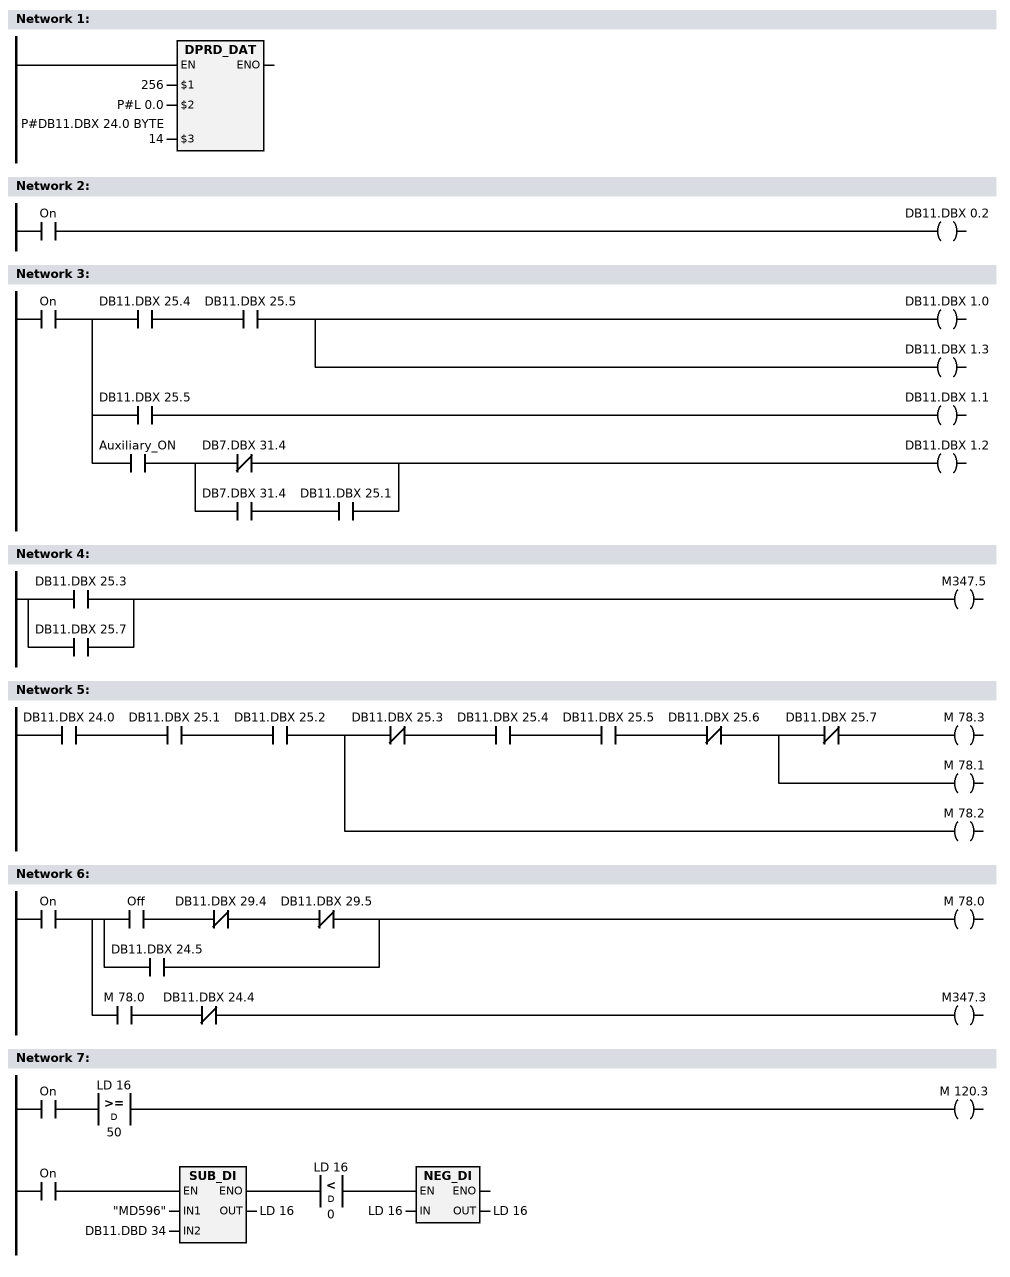
[picture p149: FC - AUTOMATIC networks 1-7]
NETWORK
TITLE =
      CALL  "DPRD_DAT" (
           $1                       := 256,
           $2                       := P#L 0.0,
           $3                       := P#DB11.DBX 24.0 BYTE 14);
      NOP   0;
NETWORK
TITLE =
      A     "On";
      =     DB11.DBX 0.2;
NETWORK
TITLE =
      A     "On";
      =     L 21.0;
      A     L 21.0;
      A     DB11.DBX 25.4;
      A     DB11.DBX 25.5;
      =     DB11.DBX 1.0;
      =     DB11.DBX 1.3;
      A     L 21.0;
      A     DB11.DBX 25.5;
      =     DB11.DBX 1.1;
      A     L 21.0;
      A     "Auxiliary_ON";
      A(;
      ON    DB7.DBX 31.4;
      O;
      A     DB7.DBX 31.4;
      A     DB11.DBX 25.1;
      );
      =     DB11.DBX 1.2;
NETWORK
TITLE =
      O     DB11.DBX 25.3;
      O     DB11.DBX 25.7;
      =     "M347.5";
NETWORK
TITLE =
      A     DB11.DBX 24.0;
      A     DB11.DBX 25.1;
      A     DB11.DBX 25.2;
      =     L 21.0;
      A     L 21.0;
      AN    DB11.DBX 25.3;
      A     DB11.DBX 25.4;
      A     DB11.DBX 25.5;
      AN    DB11.DBX 25.6;
      =     L 21.1;
      A     L 21.1;
      AN    DB11.DBX 25.7;
      =     M 78.3;
      A     L 21.1;
      BLD   102;
      =     M 78.1;
      A     L 21.0;
      BLD   102;
      =     M 78.2;
NETWORK
TITLE =
      A     "On";
      =     L 21.0;
      A     L 21.0;
      A(;
      A     "Off";
      AN    DB11.DBX 29.4;
      AN    DB11.DBX 29.5;
      O     DB11.DBX 24.5;
      );
      =     M 78.0;
      A     L 21.0;
      A     M 78.0;
      AN    DB11.DBX 24.4;
      =     "M347.3";
NETWORK
TITLE =
      A     "On";
      =     L 20.0;
      A(;
      A     L 20.0;
      JNB   M001;
      L     "MD596";
      L     DB11.DBD 34;
      -D;
      T     LD 16;
      AN    OV;
      SAVE;
      CLR;
M001: A     BR;
      );
      A(;
      L     LD 16;
      L     0;
      <D;
      );
      JNB   M002;
      L     LD 16;
      NEGD;
      T     LD 16;
M002: NOP   0;
      A     L 20.0;
      A(;
      L     LD 16;
      L     50;
      >=D;
      );
      =     M 120.3;
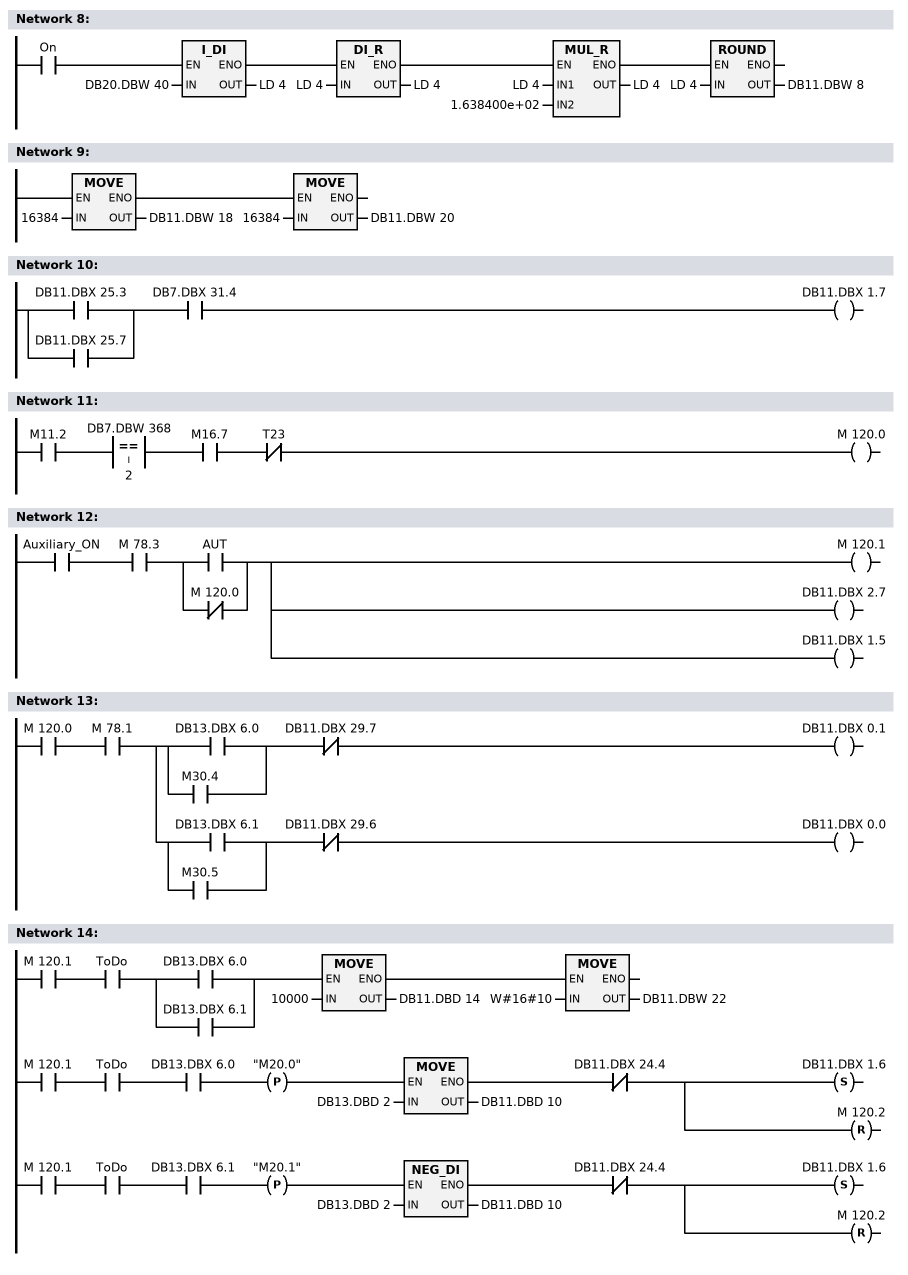
NETWORK
TITLE =
      A(;
      A(;
      A(;
      A     "On";
      JNB   M003;
      L     DB20.DBW 40;
      ITD;
      T     LD 4;
      SET;
      SAVE;
      CLR;
M003: A     BR;
      );
      JNB   M004;
      L     LD 4;
      DTR;
      T     LD 4;
      SET;
      SAVE;
      CLR;
M004: A     BR;
      );
      JNB   M005;
      L     LD 4;
      L     1.638400e+02;
      *R;
      T     LD 4;
      AN    OV;
      SAVE;
      CLR;
M005: A     BR;
      );
      JNB   M006;
      L     LD 4;
      RND;
      T     DB11.DBW 8;
M006: NOP   0;
NETWORK
TITLE =
      A(;
      L     16384;
      T     DB11.DBW 18;
      SET;
      SAVE;
      CLR;
      A     BR;
      );
      JNB   M007;
      L     16384;
      T     DB11.DBW 20;
M007: NOP   0;
NETWORK
TITLE =
      A(;
      O     DB11.DBX 25.3;
      O     DB11.DBX 25.7;
      );
      A     DB7.DBX 31.4;
      =     DB11.DBX 1.7;
NETWORK
TITLE =
      A     "M11.2";
      A(;
      L     DB7.DBW 368;
      L     2;
      ==I;
      );
      A     "M16.7";
      AN    "T23";
      =     M 120.0;
NETWORK
TITLE =
      A     "Auxiliary_ON";
      A     M 78.3;
      A(;
      O     "AUT";
      ON    M 120.0;
      );
      =     M 120.1;
      =     DB11.DBX 2.7;
      =     DB11.DBX 1.5;
NETWORK
TITLE =
      A     M 120.0;
      A     M 78.1;
      =     L 21.0;
      A     L 21.0;
      A(;
      O     DB13.DBX 6.0;
      O     "M30.4";
      );
      AN    DB11.DBX 29.7;
      =     DB11.DBX 0.1;
      A     L 21.0;
      A(;
      O     DB13.DBX 6.1;
      O     "M30.5";
      );
      AN    DB11.DBX 29.6;
      =     DB11.DBX 0.0;
NETWORK
TITLE =
      A     M 120.1;
      A     "ToDo";
      =     L 21.0;
      A(;
      A     L 21.0;
      A(;
      O     DB13.DBX 6.0;
      O     DB13.DBX 6.1;
      );
      JNB   M008;
      L     10000;
      T     DB11.DBD 14;
      SET;
      SAVE;
      CLR;
M008: A     BR;
      );
      JNB   M009;
      L     W#16#10;
      T     DB11.DBW 22;
M009: NOP   0;
      A(;
      A     L 21.0;
      A     DB13.DBX 6.0;
      FP    "M20.0";
      JNB   M010;
      L     DB13.DBD 2;
      T     DB11.DBD 10;
      SET;
      SAVE;
      CLR;
M010: A     BR;
      );
      AN    DB11.DBX 24.4;
      S     DB11.DBX 1.6;
      R     M 120.2;
      A(;
      A     L 21.0;
      A     DB13.DBX 6.1;
      FP    "M20.1";
      JNB   M011;
      L     DB13.DBD 2;
      NEGD;
      T     DB11.DBD 10;
      AN    OV;
      SAVE;
      CLR;
M011: A     BR;
      );
      AN    DB11.DBX 24.4;
      S     DB11.DBX 1.6;
      R     M 120.2;
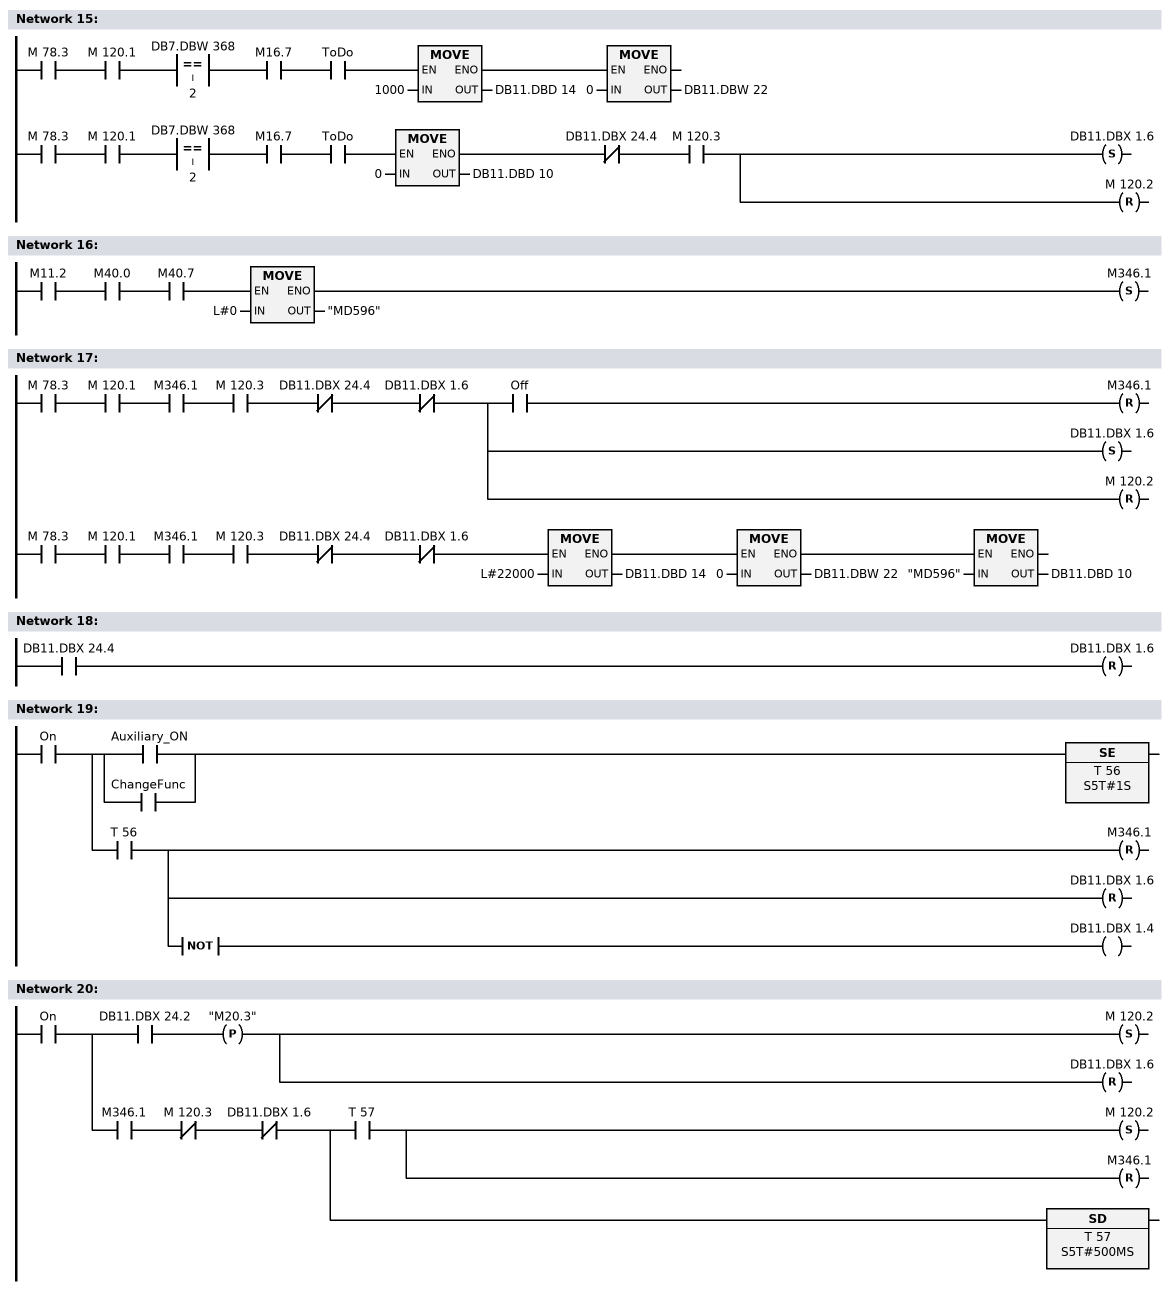
NETWORK
TITLE =
      A     M 78.3;
      A     M 120.1;
      A(;
      L     DB7.DBW 368;
      L     2;
      ==I;
      );
      A     "M16.7";
      =     L 21.0;
      A(;
      A     L 21.0;
      A     "ToDo";
      JNB   M012;
      L     1000;
      T     DB11.DBD 14;
      SET;
      SAVE;
      CLR;
M012: A     BR;
      );
      JNB   M013;
      L     0;
      T     DB11.DBW 22;
M013: NOP   0;
      A(;
      A     L 21.0;
      A     "ToDo";
      JNB   M014;
      L     0;
      T     DB11.DBD 10;
      SET;
      SAVE;
      CLR;
M014: A     BR;
      );
      AN    DB11.DBX 24.4;
      A     M 120.3;
      S     DB11.DBX 1.6;
      R     M 120.2;
NETWORK
TITLE =
      A     "M11.2";
      A     "M40.0";
      A     "M40.7";
      JNB   M015;
      L     L#0;
      T     "MD596";
      SET;
      SAVE;
      CLR;
M015: A     BR;
      S     "M346.1";
NETWORK
TITLE =
      A     M 78.3;
      A     M 120.1;
      A     "M346.1";
      A     M 120.3;
      AN    DB11.DBX 24.4;
      AN    DB11.DBX 1.6;
      =     L 21.0;
      A(;
      A(;
      A     L 21.0;
      JNB   M016;
      L     L#22000;
      T     DB11.DBD 14;
      SET;
      SAVE;
      CLR;
M016: A     BR;
      );
      JNB   M017;
      L     0;
      T     DB11.DBW 22;
      SET;
      SAVE;
      CLR;
M017: A     BR;
      );
      JNB   M018;
      L     "MD596";
      T     DB11.DBD 10;
M018: NOP   0;
      A     L 21.0;
      A     "Off";
      R     "M346.1";
      A     L 21.0;
      BLD   102;
      S     DB11.DBX 1.6;
      A     L 21.0;
      BLD   102;
      R     M 120.2;
NETWORK
TITLE =
      A     DB11.DBX 24.4;
      R     DB11.DBX 1.6;
NETWORK
TITLE =
      A     "On";
      =     L 21.0;
      A     L 21.0;
      A(;
      O     "Auxiliary_ON";
      O     "ChangeFunc";
      );
      L     S5T#1S;
      SE    T 56;
      A     L 21.0;
      A     T 56;
      =     L 21.1;
      A     L 21.1;
      BLD   102;
      R     "M346.1";
      A     L 21.1;
      BLD   102;
      R     DB11.DBX 1.6;
      A     L 21.1;
      NOT;
      =     DB11.DBX 1.4;
NETWORK
TITLE =
      A     "On";
      =     L 21.0;
      A     L 21.0;
      A     DB11.DBX 24.2;
      FP    "M20.3";
      S     M 120.2;
      R     DB11.DBX 1.6;
      A     L 21.0;
      A     "M346.1";
      AN    M 120.3;
      AN    DB11.DBX 1.6;
      =     L 21.1;
      A     L 21.1;
      A     T 57;
      S     M 120.2;
      R     "M346.1";
      A     L 21.1;
      BLD   102;
      L     S5T#500MS;
      SD    T 57;
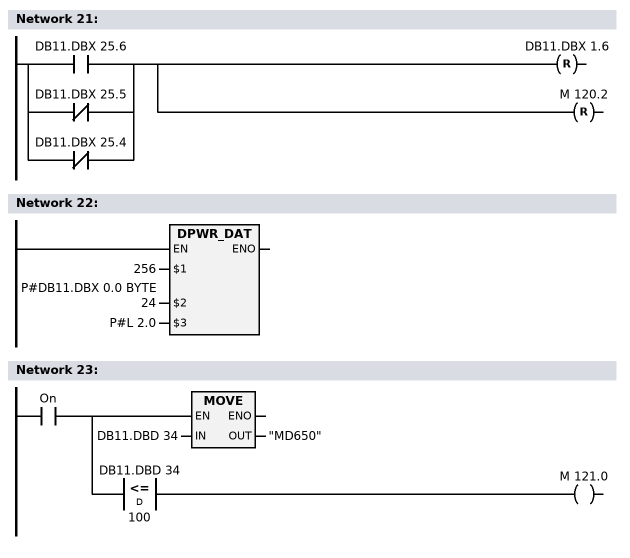
NETWORK
TITLE =
      O     DB11.DBX 25.6;
      ON    DB11.DBX 25.5;
      ON    DB11.DBX 25.4;
      R     DB11.DBX 1.6;
      R     M 120.2;
NETWORK
TITLE =
      CALL  "DPWR_DAT" (
           $1                       := 256,
           $2                       := P#DB11.DBX 0.0 BYTE 24,
           $3                       := P#L 2.0);
      NOP   0;
NETWORK
TITLE =
      A     "On";
      =     L 20.0;
      A     L 20.0;
      JNB   M019;
      L     DB11.DBD 34;
      T     "MD650";
M019: NOP   0;
      A     L 20.0;
      A(;
      L     DB11.DBD 34;
      L     100;
      <=D;
      );
      =     M 121.0;
END_FUNCTION

FUNCTION FC 25 : VOID
VERSION : 0.1
BEGIN
// (block stored without names or comments; labels and parameter names are numbered)
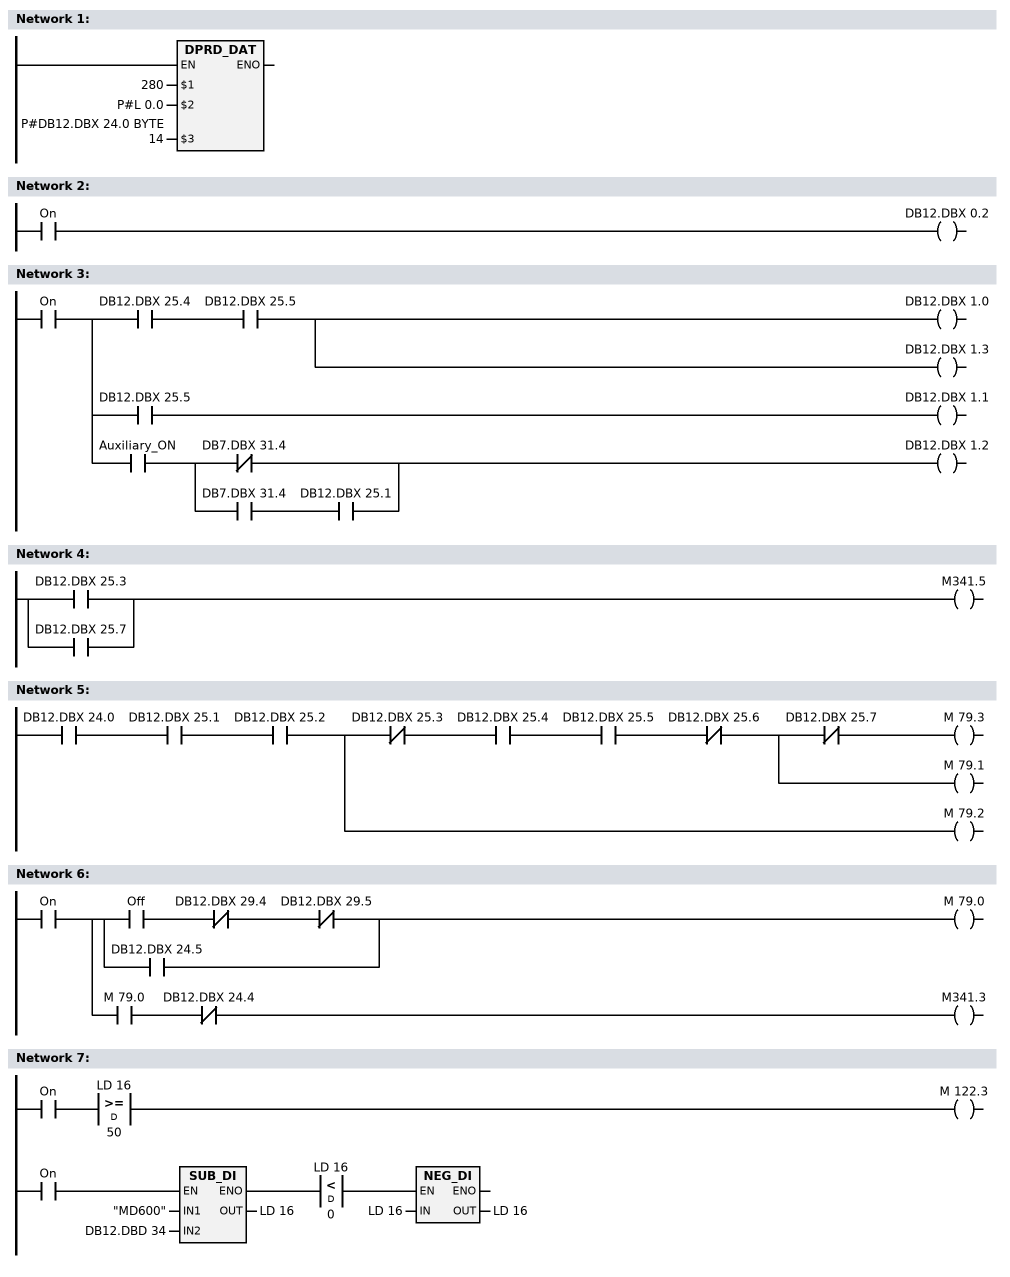
NETWORK
TITLE =
      CALL  "DPRD_DAT" (
           $1                       := 280,
           $2                       := P#L 0.0,
           $3                       := P#DB12.DBX 24.0 BYTE 14);
      NOP   0;
NETWORK
TITLE =
      A     "On";
      =     DB12.DBX 0.2;
NETWORK
TITLE =
      A     "On";
      =     L 21.0;
      A     L 21.0;
      A     DB12.DBX 25.4;
      A     DB12.DBX 25.5;
      =     DB12.DBX 1.0;
      =     DB12.DBX 1.3;
      A     L 21.0;
      A     DB12.DBX 25.5;
      =     DB12.DBX 1.1;
      A     L 21.0;
      A     "Auxiliary_ON";
      A(;
      ON    DB7.DBX 31.4;
      O;
      A     DB7.DBX 31.4;
      A     DB12.DBX 25.1;
      );
      =     DB12.DBX 1.2;
NETWORK
TITLE =
      O     DB12.DBX 25.3;
      O     DB12.DBX 25.7;
      =     "M341.5";
NETWORK
TITLE =
      A     DB12.DBX 24.0;
      A     DB12.DBX 25.1;
      A     DB12.DBX 25.2;
      =     L 21.0;
      A     L 21.0;
      AN    DB12.DBX 25.3;
      A     DB12.DBX 25.4;
      A     DB12.DBX 25.5;
      AN    DB12.DBX 25.6;
      =     L 21.1;
      A     L 21.1;
      AN    DB12.DBX 25.7;
      =     M 79.3;
      A     L 21.1;
      BLD   102;
      =     M 79.1;
      A     L 21.0;
      BLD   102;
      =     M 79.2;
NETWORK
TITLE =
      A     "On";
      =     L 21.0;
      A     L 21.0;
      A(;
      A     "Off";
      AN    DB12.DBX 29.4;
      AN    DB12.DBX 29.5;
      O     DB12.DBX 24.5;
      );
      =     M 79.0;
      A     L 21.0;
      A     M 79.0;
      AN    DB12.DBX 24.4;
      =     "M341.3";
NETWORK
TITLE =
      A     "On";
      =     L 20.0;
      A(;
      A     L 20.0;
      JNB   M001;
      L     "MD600";
      L     DB12.DBD 34;
      -D;
      T     LD 16;
      AN    OV;
      SAVE;
      CLR;
M001: A     BR;
      );
      A(;
      L     LD 16;
      L     0;
      <D;
      );
      JNB   M002;
      L     LD 16;
      NEGD;
      T     LD 16;
M002: NOP   0;
      A     L 20.0;
      A(;
      L     LD 16;
      L     50;
      >=D;
      );
      =     M 122.3;
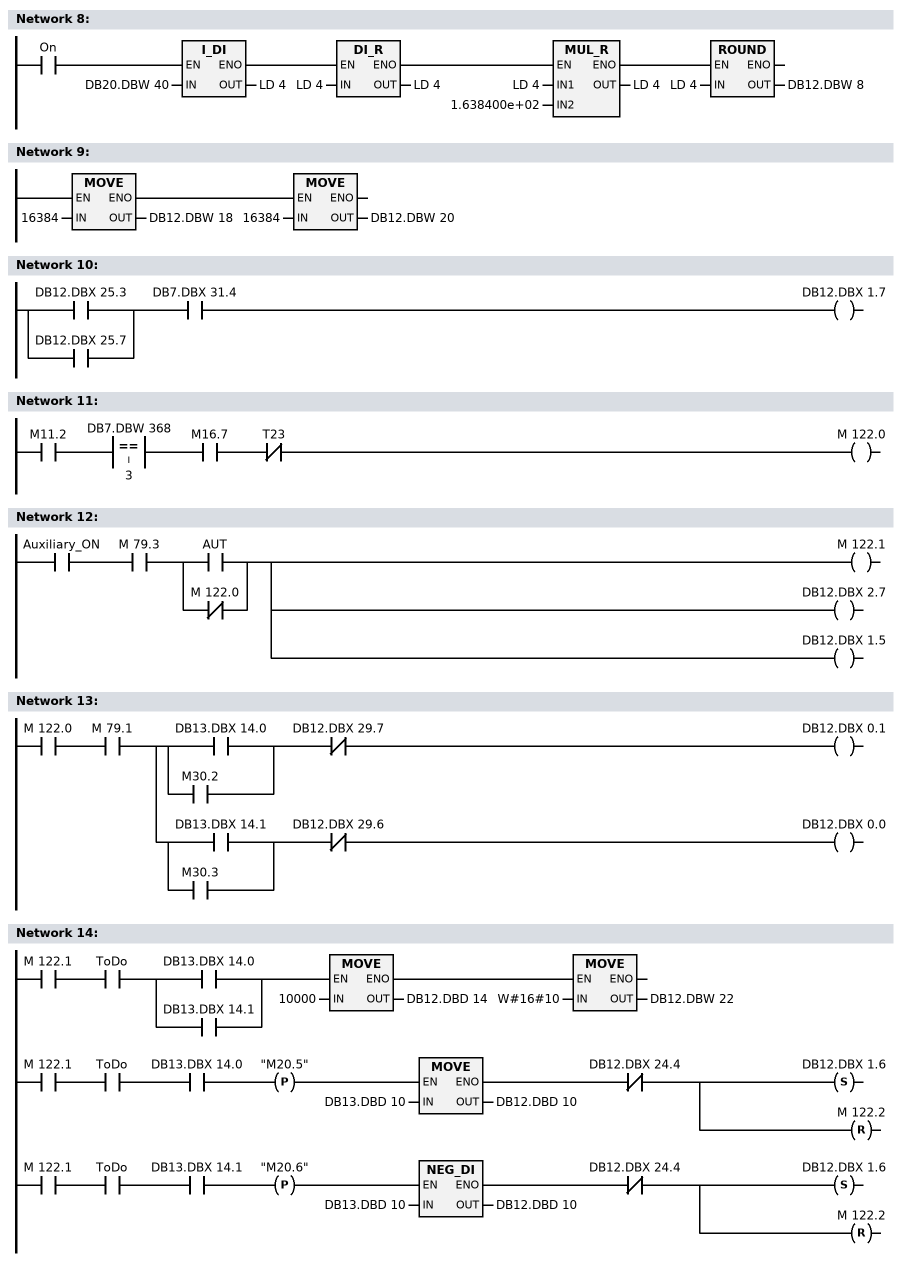
NETWORK
TITLE =
      A(;
      A(;
      A(;
      A     "On";
      JNB   M003;
      L     DB20.DBW 40;
      ITD;
      T     LD 4;
      SET;
      SAVE;
      CLR;
M003: A     BR;
      );
      JNB   M004;
      L     LD 4;
      DTR;
      T     LD 4;
      SET;
      SAVE;
      CLR;
M004: A     BR;
      );
      JNB   M005;
      L     LD 4;
      L     1.638400e+02;
      *R;
      T     LD 4;
      AN    OV;
      SAVE;
      CLR;
M005: A     BR;
      );
      JNB   M006;
      L     LD 4;
      RND;
      T     DB12.DBW 8;
M006: NOP   0;
NETWORK
TITLE =
      A(;
      L     16384;
      T     DB12.DBW 18;
      SET;
      SAVE;
      CLR;
      A     BR;
      );
      JNB   M007;
      L     16384;
      T     DB12.DBW 20;
M007: NOP   0;
NETWORK
TITLE =
      A(;
      O     DB12.DBX 25.3;
      O     DB12.DBX 25.7;
      );
      A     DB7.DBX 31.4;
      =     DB12.DBX 1.7;
NETWORK
TITLE =
      A     "M11.2";
      A(;
      L     DB7.DBW 368;
      L     3;
      ==I;
      );
      A     "M16.7";
      AN    "T23";
      =     M 122.0;
NETWORK
TITLE =
      A     "Auxiliary_ON";
      A     M 79.3;
      A(;
      O     "AUT";
      ON    M 122.0;
      );
      =     M 122.1;
      =     DB12.DBX 2.7;
      =     DB12.DBX 1.5;
NETWORK
TITLE =
      A     M 122.0;
      A     M 79.1;
      =     L 21.0;
      A     L 21.0;
      A(;
      O     DB13.DBX 14.0;
      O     "M30.2";
      );
      AN    DB12.DBX 29.7;
      =     DB12.DBX 0.1;
      A     L 21.0;
      A(;
      O     DB13.DBX 14.1;
      O     "M30.3";
      );
      AN    DB12.DBX 29.6;
      =     DB12.DBX 0.0;
NETWORK
TITLE =
      A     M 122.1;
      A     "ToDo";
      =     L 21.0;
      A(;
      A     L 21.0;
      A(;
      O     DB13.DBX 14.0;
      O     DB13.DBX 14.1;
      );
      JNB   M008;
      L     10000;
      T     DB12.DBD 14;
      SET;
      SAVE;
      CLR;
M008: A     BR;
      );
      JNB   M009;
      L     W#16#10;
      T     DB12.DBW 22;
M009: NOP   0;
      A(;
      A     L 21.0;
      A     DB13.DBX 14.0;
      FP    "M20.5";
      JNB   M010;
      L     DB13.DBD 10;
      T     DB12.DBD 10;
      SET;
      SAVE;
      CLR;
M010: A     BR;
      );
      AN    DB12.DBX 24.4;
      S     DB12.DBX 1.6;
      R     M 122.2;
      A(;
      A     L 21.0;
      A     DB13.DBX 14.1;
      FP    "M20.6";
      JNB   M011;
      L     DB13.DBD 10;
      NEGD;
      T     DB12.DBD 10;
      AN    OV;
      SAVE;
      CLR;
M011: A     BR;
      );
      AN    DB12.DBX 24.4;
      S     DB12.DBX 1.6;
      R     M 122.2;
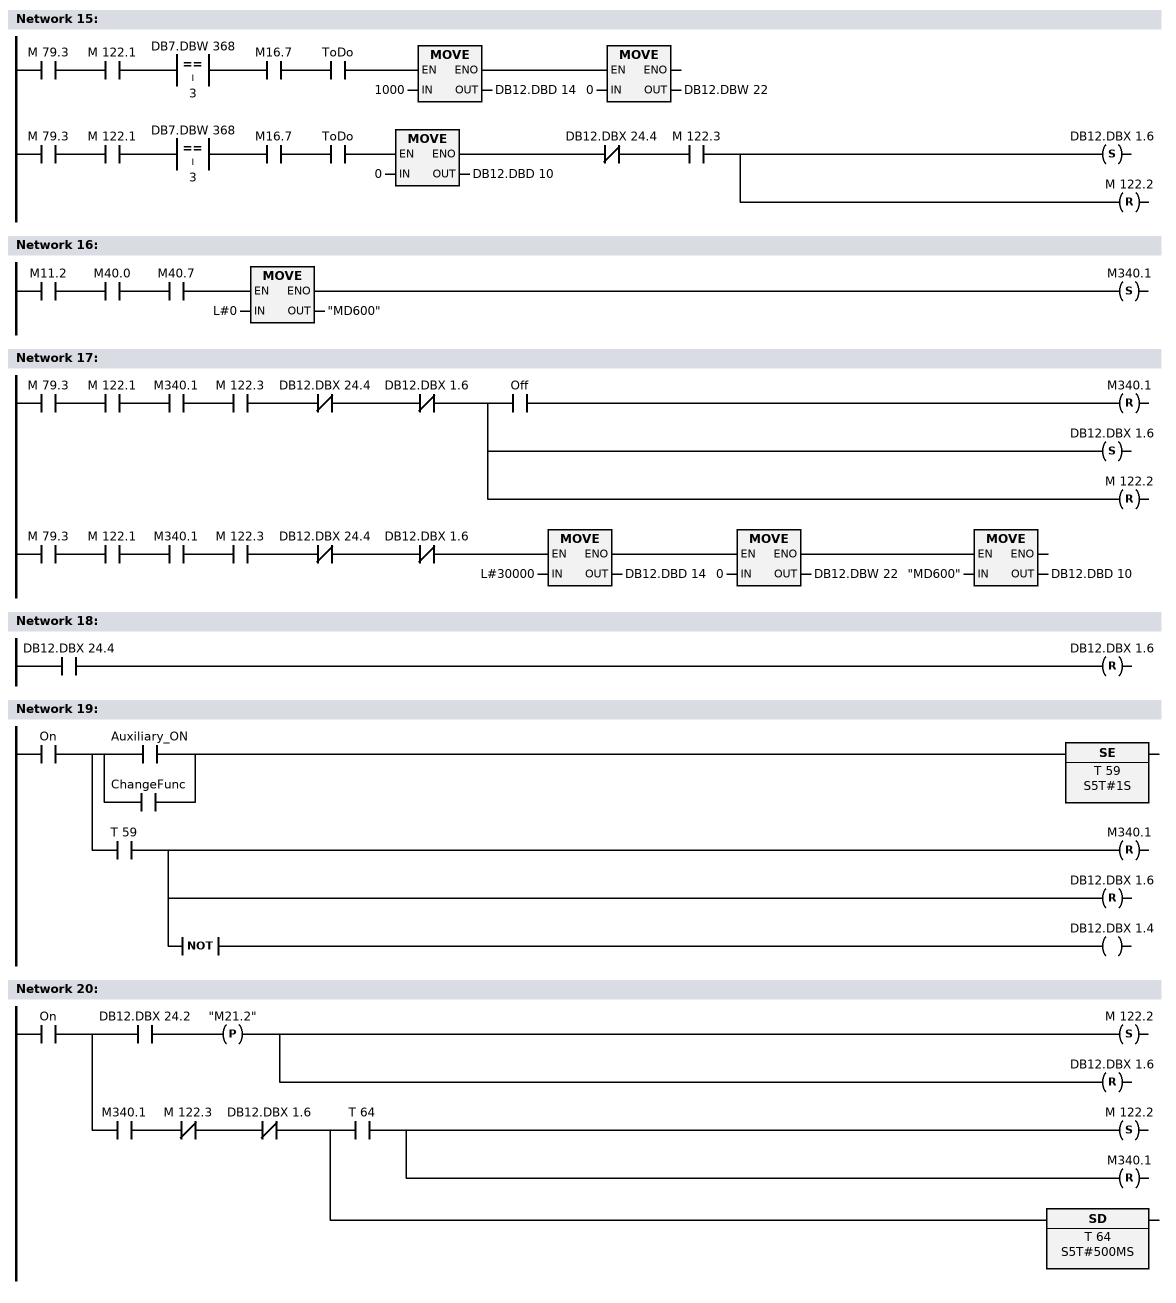
NETWORK
TITLE =
      A     M 79.3;
      A     M 122.1;
      A(;
      L     DB7.DBW 368;
      L     3;
      ==I;
      );
      A     "M16.7";
      =     L 21.0;
      A(;
      A     L 21.0;
      A     "ToDo";
      JNB   M012;
      L     1000;
      T     DB12.DBD 14;
      SET;
      SAVE;
      CLR;
M012: A     BR;
      );
      JNB   M013;
      L     0;
      T     DB12.DBW 22;
M013: NOP   0;
      A(;
      A     L 21.0;
      A     "ToDo";
      JNB   M014;
      L     0;
      T     DB12.DBD 10;
      SET;
      SAVE;
      CLR;
M014: A     BR;
      );
      AN    DB12.DBX 24.4;
      A     M 122.3;
      S     DB12.DBX 1.6;
      R     M 122.2;
NETWORK
TITLE =
      A     "M11.2";
      A     "M40.0";
      A     "M40.7";
      JNB   M015;
      L     L#0;
      T     "MD600";
      SET;
      SAVE;
      CLR;
M015: A     BR;
      S     "M340.1";
NETWORK
TITLE =
      A     M 79.3;
      A     M 122.1;
      A     "M340.1";
      A     M 122.3;
      AN    DB12.DBX 24.4;
      AN    DB12.DBX 1.6;
      =     L 21.0;
      A(;
      A(;
      A     L 21.0;
      JNB   M016;
      L     L#30000;
      T     DB12.DBD 14;
      SET;
      SAVE;
      CLR;
M016: A     BR;
      );
      JNB   M017;
      L     0;
      T     DB12.DBW 22;
      SET;
      SAVE;
      CLR;
M017: A     BR;
      );
      JNB   M018;
      L     "MD600";
      T     DB12.DBD 10;
M018: NOP   0;
      A     L 21.0;
      A     "Off";
      R     "M340.1";
      A     L 21.0;
      BLD   102;
      S     DB12.DBX 1.6;
      A     L 21.0;
      BLD   102;
      R     M 122.2;
NETWORK
TITLE =
      A     DB12.DBX 24.4;
      R     DB12.DBX 1.6;
NETWORK
TITLE =
      A     "On";
      =     L 21.0;
      A     L 21.0;
      A(;
      O     "Auxiliary_ON";
      O     "ChangeFunc";
      );
      L     S5T#1S;
      SE    T 59;
      A     L 21.0;
      A     T 59;
      =     L 21.1;
      A     L 21.1;
      BLD   102;
      R     "M340.1";
      A     L 21.1;
      BLD   102;
      R     DB12.DBX 1.6;
      A     L 21.1;
      NOT;
      =     DB12.DBX 1.4;
NETWORK
TITLE =
      A     "On";
      =     L 21.0;
      A     L 21.0;
      A     DB12.DBX 24.2;
      FP    "M21.2";
      S     M 122.2;
      R     DB12.DBX 1.6;
      A     L 21.0;
      A     "M340.1";
      AN    M 122.3;
      AN    DB12.DBX 1.6;
      =     L 21.1;
      A     L 21.1;
      A     T 64;
      S     M 122.2;
      R     "M340.1";
      A     L 21.1;
      BLD   102;
      L     S5T#500MS;
      SD    T 64;
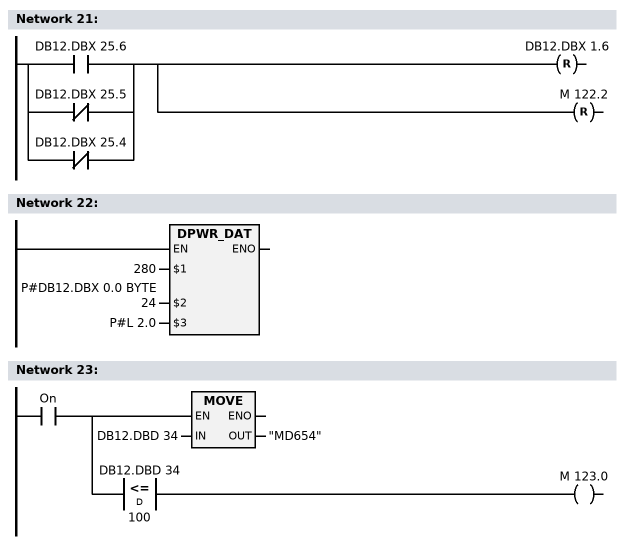
NETWORK
TITLE =
      O     DB12.DBX 25.6;
      ON    DB12.DBX 25.5;
      ON    DB12.DBX 25.4;
      R     DB12.DBX 1.6;
      R     M 122.2;
NETWORK
TITLE =
      CALL  "DPWR_DAT" (
           $1                       := 280,
           $2                       := P#DB12.DBX 0.0 BYTE 24,
           $3                       := P#L 2.0);
      NOP   0;
NETWORK
TITLE =
      A     "On";
      =     L 20.0;
      A     L 20.0;
      JNB   M019;
      L     DB12.DBD 34;
      T     "MD654";
M019: NOP   0;
      A     L 20.0;
      A(;
      L     DB12.DBD 34;
      L     100;
      <=D;
      );
      =     M 123.0;
END_FUNCTION

FUNCTION "FC50 - TEACH-IN" : VOID	// FC 50
VERSION : 0.1
BEGIN
// (block stored without names or comments; labels and parameter names are numbered)
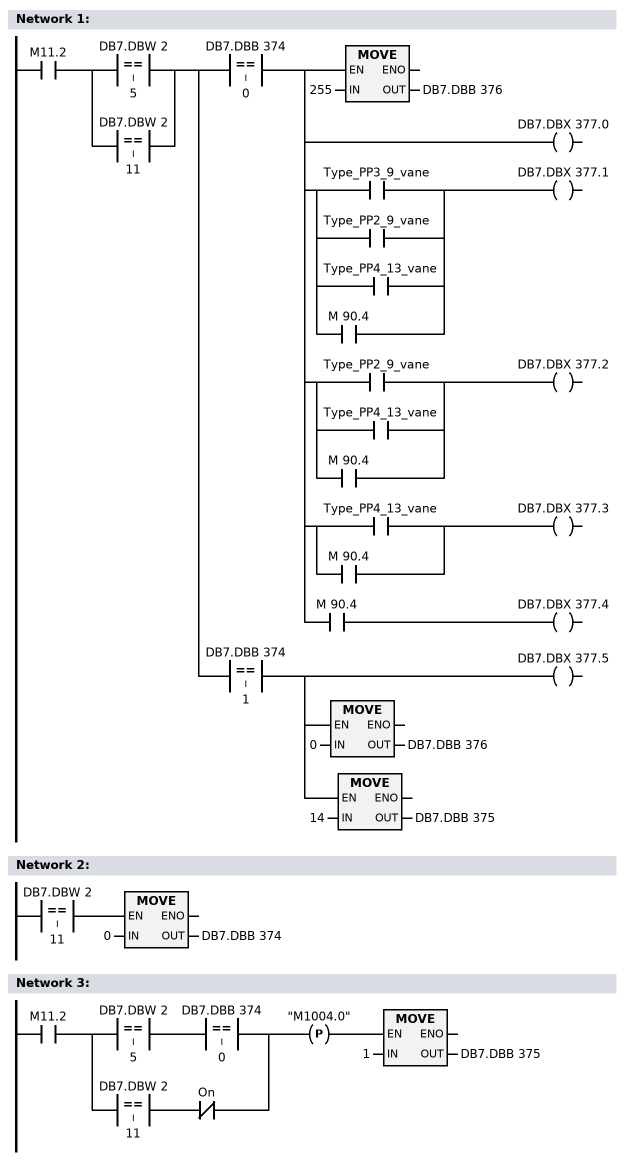
NETWORK
TITLE =
      A     "M11.2";
      A(;
      O(;
      L     DB7.DBW 2;
      L     5;
      ==I;
      );
      O(;
      L     DB7.DBW 2;
      L     11;
      ==I;
      );
      );
      =     L 8.0;
      A     L 8.0;
      A(;
      L     DB7.DBB 374;
      L     0;
      ==I;
      );
      =     L 8.1;
      A     L 8.1;
      JNB   M001;
      L     255;
      T     DB7.DBB 376;
M001: NOP   0;
      A     L 8.1;
      BLD   102;
      =     DB7.DBX 377.0;
      A     L 8.1;
      A(;
      O     "Type_PP3_9_vane";
      O     "Type_PP2_9_vane";
      O     "Type_PP4_13_vane";
      O     M 90.4;
      );
      =     DB7.DBX 377.1;
      A     L 8.1;
      A(;
      O     "Type_PP2_9_vane";
      O     "Type_PP4_13_vane";
      O     M 90.4;
      );
      =     DB7.DBX 377.2;
      A     L 8.1;
      A(;
      O     "Type_PP4_13_vane";
      O     M 90.4;
      );
      =     DB7.DBX 377.3;
      A     L 8.1;
      A     M 90.4;
      =     DB7.DBX 377.4;
      A     L 8.0;
      A(;
      L     DB7.DBB 374;
      L     1;
      ==I;
      );
      =     L 8.1;
      A     L 8.1;
      BLD   102;
      =     DB7.DBX 377.5;
      A     L 8.1;
      JNB   M002;
      L     0;
      T     DB7.DBB 376;
M002: NOP   0;
      A     L 8.1;
      JNB   M003;
      L     14;
      T     DB7.DBB 375;
M003: NOP   0;
NETWORK
TITLE =
      A(;
      L     DB7.DBW 2;
      L     11;
      ==I;
      );
      JNB   M004;
      L     0;
      T     DB7.DBB 374;
M004: NOP   0;
NETWORK
TITLE =
      A     "M11.2";
      A(;
      A(;
      L     DB7.DBW 2;
      L     5;
      ==I;
      );
      A(;
      L     DB7.DBB 374;
      L     0;
      ==I;
      );
      O;
      A(;
      L     DB7.DBW 2;
      L     11;
      ==I;
      );
      AN    "On";
      );
      FP    "M1004.0";
      JNB   M005;
      L     1;
      T     DB7.DBB 375;
M005: NOP   0;
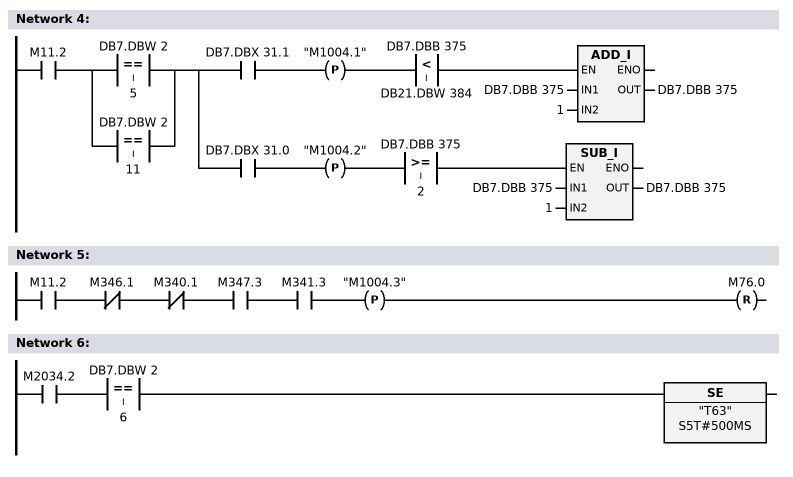
NETWORK
TITLE =
      A     "M11.2";
      A(;
      O(;
      L     DB7.DBW 2;
      L     5;
      ==I;
      );
      O(;
      L     DB7.DBW 2;
      L     11;
      ==I;
      );
      );
      =     L 8.0;
      A     L 8.0;
      A     DB7.DBX 31.1;
      FP    "M1004.1";
      A(;
      L     DB7.DBB 375;
      L     DB21.DBW 384;
      <I;
      );
      JNB   M006;
      L     DB7.DBB 375;
      L     1;
      +I;
      T     DB7.DBB 375;
M006: NOP   0;
      A     L 8.0;
      A     DB7.DBX 31.0;
      FP    "M1004.2";
      A(;
      L     DB7.DBB 375;
      L     2;
      >=I;
      );
      JNB   M007;
      L     DB7.DBB 375;
      L     1;
      -I;
      T     DB7.DBB 375;
M007: NOP   0;
NETWORK
TITLE =
      A     "M11.2";
      AN    "M346.1";
      AN    "M340.1";
      A     "M347.3";
      A     "M341.3";
      FP    "M1004.3";
      R     "M76.0";
NETWORK
TITLE =
      A     "M2034.2";
      A(;
      L     DB7.DBW 2;
      L     6;
      ==I;
      );
      L     S5T#500MS;
      SE    "T63";
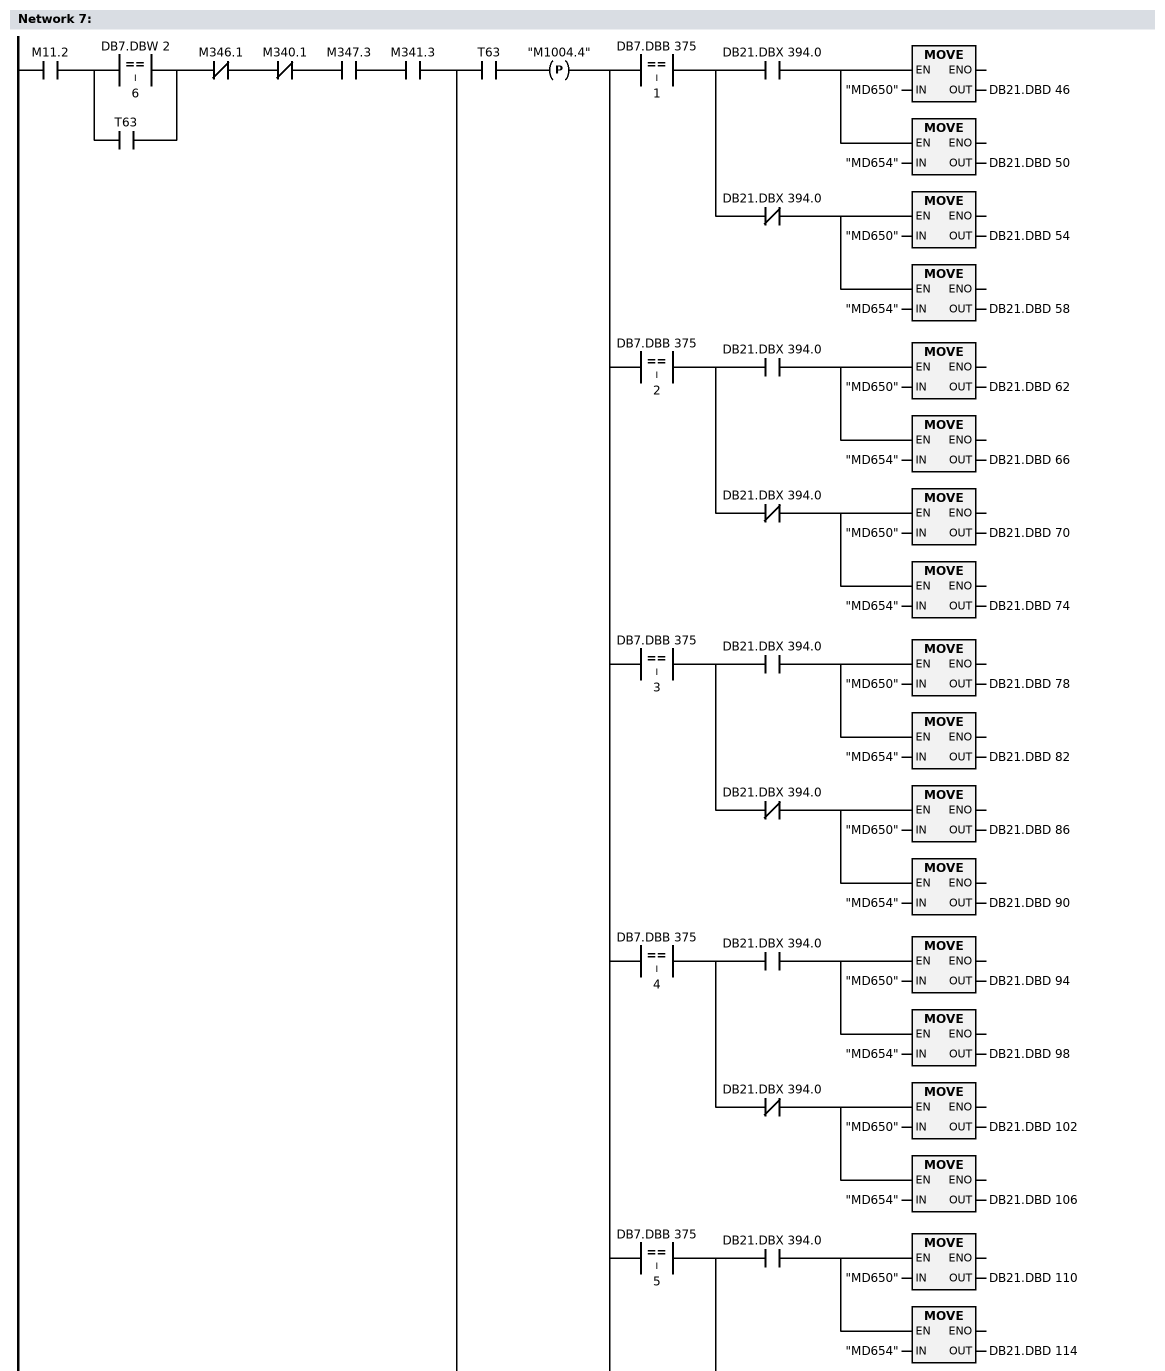
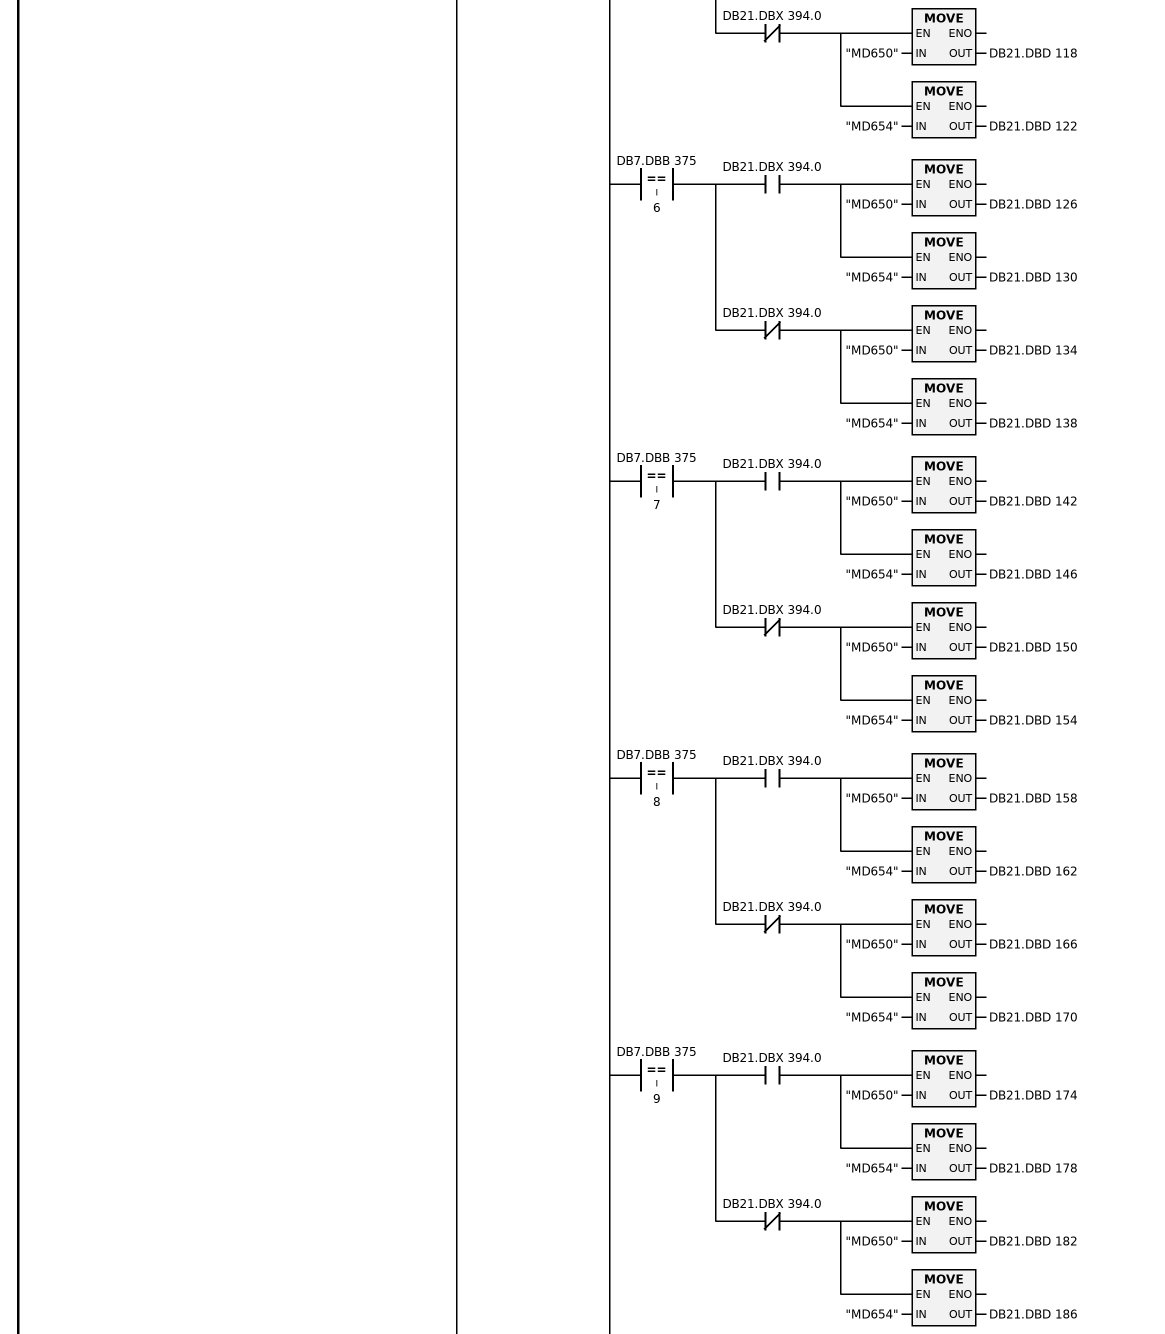
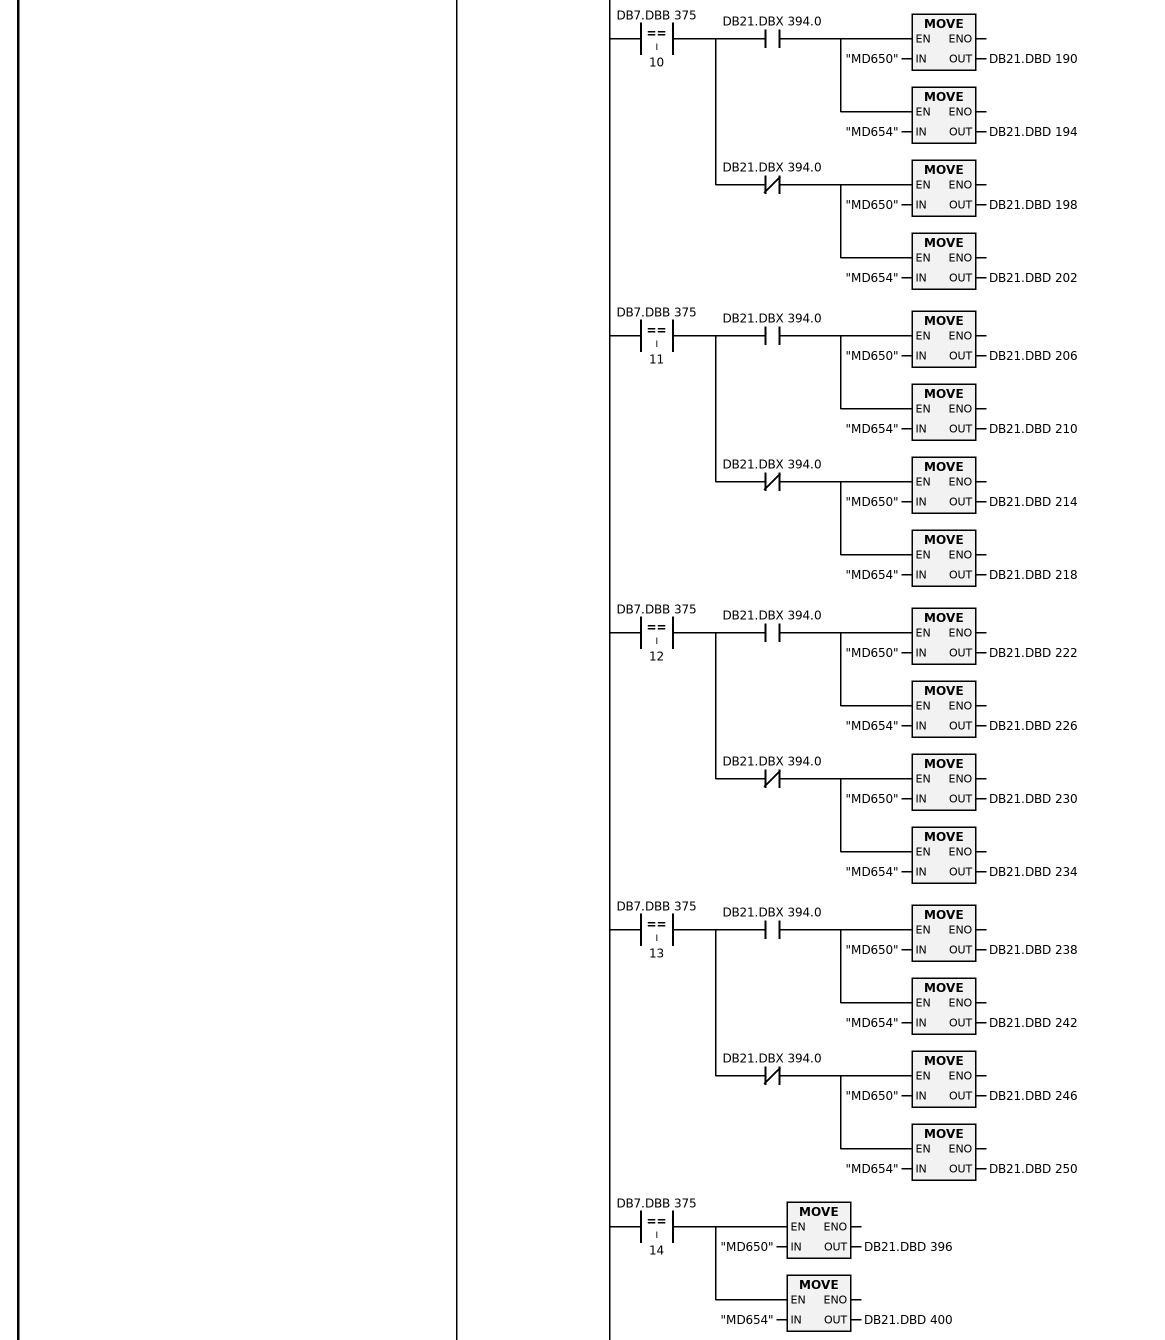
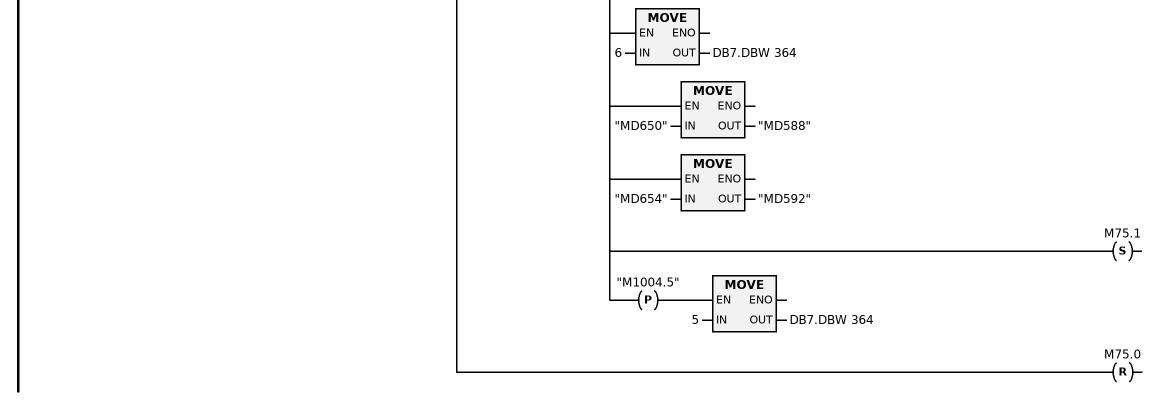
NETWORK
TITLE =
      A     "M11.2";
      A(;
      O(;
      L     DB7.DBW 2;
      L     6;
      ==I;
      );
      O     "T63";
      );
      AN    "M346.1";
      AN    "M340.1";
      A     "M347.3";
      A     "M341.3";
      =     L 8.0;
      A     L 8.0;
      A     "T63";
      FP    "M1004.4";
      =     L 8.1;
      A     L 8.1;
      A(;
      L     DB7.DBB 375;
      L     1;
      ==I;
      );
      =     L 8.2;
      A     L 8.2;
      A     DB21.DBX 394.0;
      =     L 8.3;
      A     L 8.3;
      JNB   M008;
      L     "MD650";
      T     DB21.DBD 46;
M008: NOP   0;
      A     L 8.3;
      JNB   M009;
      L     "MD654";
      T     DB21.DBD 50;
M009: NOP   0;
      A     L 8.2;
      AN    DB21.DBX 394.0;
      =     L 8.3;
      A     L 8.3;
      JNB   M010;
      L     "MD650";
      T     DB21.DBD 54;
M010: NOP   0;
      A     L 8.3;
      JNB   M011;
      L     "MD654";
      T     DB21.DBD 58;
M011: NOP   0;
      A     L 8.1;
      A(;
      L     DB7.DBB 375;
      L     2;
      ==I;
      );
      =     L 8.2;
      A     L 8.2;
      A     DB21.DBX 394.0;
      =     L 8.3;
      A     L 8.3;
      JNB   M012;
      L     "MD650";
      T     DB21.DBD 62;
M012: NOP   0;
      A     L 8.3;
      JNB   M013;
      L     "MD654";
      T     DB21.DBD 66;
M013: NOP   0;
      A     L 8.2;
      AN    DB21.DBX 394.0;
      =     L 8.3;
      A     L 8.3;
      JNB   M014;
      L     "MD650";
      T     DB21.DBD 70;
M014: NOP   0;
      A     L 8.3;
      JNB   M015;
      L     "MD654";
      T     DB21.DBD 74;
M015: NOP   0;
      A     L 8.1;
      A(;
      L     DB7.DBB 375;
      L     3;
      ==I;
      );
      =     L 8.2;
      A     L 8.2;
      A     DB21.DBX 394.0;
      =     L 8.3;
      A     L 8.3;
      JNB   M016;
      L     "MD650";
      T     DB21.DBD 78;
M016: NOP   0;
      A     L 8.3;
      JNB   M017;
      L     "MD654";
      T     DB21.DBD 82;
M017: NOP   0;
      A     L 8.2;
      AN    DB21.DBX 394.0;
      =     L 8.3;
      A     L 8.3;
      JNB   M018;
      L     "MD650";
      T     DB21.DBD 86;
M018: NOP   0;
      A     L 8.3;
      JNB   M019;
      L     "MD654";
      T     DB21.DBD 90;
M019: NOP   0;
      A     L 8.1;
      A(;
      L     DB7.DBB 375;
      L     4;
      ==I;
      );
      =     L 8.2;
      A     L 8.2;
      A     DB21.DBX 394.0;
      =     L 8.3;
      A     L 8.3;
      JNB   M020;
      L     "MD650";
      T     DB21.DBD 94;
M020: NOP   0;
      A     L 8.3;
      JNB   M021;
      L     "MD654";
      T     DB21.DBD 98;
M021: NOP   0;
      A     L 8.2;
      AN    DB21.DBX 394.0;
      =     L 8.3;
      A     L 8.3;
      JNB   M022;
      L     "MD650";
      T     DB21.DBD 102;
M022: NOP   0;
      A     L 8.3;
      JNB   M023;
      L     "MD654";
      T     DB21.DBD 106;
M023: NOP   0;
      A     L 8.1;
      A(;
      L     DB7.DBB 375;
      L     5;
      ==I;
      );
      =     L 8.2;
      A     L 8.2;
      A     DB21.DBX 394.0;
      =     L 8.3;
      A     L 8.3;
      JNB   M024;
      L     "MD650";
      T     DB21.DBD 110;
M024: NOP   0;
      A     L 8.3;
      JNB   M025;
      L     "MD654";
      T     DB21.DBD 114;
M025: NOP   0;
      A     L 8.2;
      AN    DB21.DBX 394.0;
      =     L 8.3;
      A     L 8.3;
      JNB   M026;
      L     "MD650";
      T     DB21.DBD 118;
M026: NOP   0;
      A     L 8.3;
      JNB   M027;
      L     "MD654";
      T     DB21.DBD 122;
M027: NOP   0;
      A     L 8.1;
      A(;
      L     DB7.DBB 375;
      L     6;
      ==I;
      );
      =     L 8.2;
      A     L 8.2;
      A     DB21.DBX 394.0;
      =     L 8.3;
      A     L 8.3;
      JNB   M028;
      L     "MD650";
      T     DB21.DBD 126;
M028: NOP   0;
      A     L 8.3;
      JNB   M029;
      L     "MD654";
      T     DB21.DBD 130;
M029: NOP   0;
      A     L 8.2;
      AN    DB21.DBX 394.0;
      =     L 8.3;
      A     L 8.3;
      JNB   M030;
      L     "MD650";
      T     DB21.DBD 134;
M030: NOP   0;
      A     L 8.3;
      JNB   M031;
      L     "MD654";
      T     DB21.DBD 138;
M031: NOP   0;
      A     L 8.1;
      A(;
      L     DB7.DBB 375;
      L     7;
      ==I;
      );
      =     L 8.2;
      A     L 8.2;
      A     DB21.DBX 394.0;
      =     L 8.3;
      A     L 8.3;
      JNB   M032;
      L     "MD650";
      T     DB21.DBD 142;
M032: NOP   0;
      A     L 8.3;
      JNB   M033;
      L     "MD654";
      T     DB21.DBD 146;
M033: NOP   0;
      A     L 8.2;
      AN    DB21.DBX 394.0;
      =     L 8.3;
      A     L 8.3;
      JNB   M034;
      L     "MD650";
      T     DB21.DBD 150;
M034: NOP   0;
      A     L 8.3;
      JNB   M035;
      L     "MD654";
      T     DB21.DBD 154;
M035: NOP   0;
      A     L 8.1;
      A(;
      L     DB7.DBB 375;
      L     8;
      ==I;
      );
      =     L 8.2;
      A     L 8.2;
      A     DB21.DBX 394.0;
      =     L 8.3;
      A     L 8.3;
      JNB   M036;
      L     "MD650";
      T     DB21.DBD 158;
M036: NOP   0;
      A     L 8.3;
      JNB   M037;
      L     "MD654";
      T     DB21.DBD 162;
M037: NOP   0;
      A     L 8.2;
      AN    DB21.DBX 394.0;
      =     L 8.3;
      A     L 8.3;
      JNB   M038;
      L     "MD650";
      T     DB21.DBD 166;
M038: NOP   0;
      A     L 8.3;
      JNB   M039;
      L     "MD654";
      T     DB21.DBD 170;
M039: NOP   0;
      A     L 8.1;
      A(;
      L     DB7.DBB 375;
      L     9;
      ==I;
      );
      =     L 8.2;
      A     L 8.2;
      A     DB21.DBX 394.0;
      =     L 8.3;
      A     L 8.3;
      JNB   M040;
      L     "MD650";
      T     DB21.DBD 174;
M040: NOP   0;
      A     L 8.3;
      JNB   M041;
      L     "MD654";
      T     DB21.DBD 178;
M041: NOP   0;
      A     L 8.2;
      AN    DB21.DBX 394.0;
      =     L 8.3;
      A     L 8.3;
      JNB   M042;
      L     "MD650";
      T     DB21.DBD 182;
M042: NOP   0;
      A     L 8.3;
      JNB   M043;
      L     "MD654";
      T     DB21.DBD 186;
M043: NOP   0;
      A     L 8.1;
      A(;
      L     DB7.DBB 375;
      L     10;
      ==I;
      );
      =     L 8.2;
      A     L 8.2;
      A     DB21.DBX 394.0;
      =     L 8.3;
      A     L 8.3;
      JNB   M044;
      L     "MD650";
      T     DB21.DBD 190;
M044: NOP   0;
      A     L 8.3;
      JNB   M045;
      L     "MD654";
      T     DB21.DBD 194;
M045: NOP   0;
      A     L 8.2;
      AN    DB21.DBX 394.0;
      =     L 8.3;
      A     L 8.3;
      JNB   M046;
      L     "MD650";
      T     DB21.DBD 198;
M046: NOP   0;
      A     L 8.3;
      JNB   M047;
      L     "MD654";
      T     DB21.DBD 202;
M047: NOP   0;
      A     L 8.1;
      A(;
      L     DB7.DBB 375;
      L     11;
      ==I;
      );
      =     L 8.2;
      A     L 8.2;
      A     DB21.DBX 394.0;
      =     L 8.3;
      A     L 8.3;
      JNB   M048;
      L     "MD650";
      T     DB21.DBD 206;
M048: NOP   0;
      A     L 8.3;
      JNB   M049;
      L     "MD654";
      T     DB21.DBD 210;
M049: NOP   0;
      A     L 8.2;
      AN    DB21.DBX 394.0;
      =     L 8.3;
      A     L 8.3;
      JNB   M050;
      L     "MD650";
      T     DB21.DBD 214;
M050: NOP   0;
      A     L 8.3;
      JNB   M051;
      L     "MD654";
      T     DB21.DBD 218;
M051: NOP   0;
      A     L 8.1;
      A(;
      L     DB7.DBB 375;
      L     12;
      ==I;
      );
      =     L 8.2;
      A     L 8.2;
      A     DB21.DBX 394.0;
      =     L 8.3;
      A     L 8.3;
      JNB   M052;
      L     "MD650";
      T     DB21.DBD 222;
M052: NOP   0;
      A     L 8.3;
      JNB   M053;
      L     "MD654";
      T     DB21.DBD 226;
M053: NOP   0;
      A     L 8.2;
      AN    DB21.DBX 394.0;
      =     L 8.3;
      A     L 8.3;
      JNB   M054;
      L     "MD650";
      T     DB21.DBD 230;
M054: NOP   0;
      A     L 8.3;
      JNB   M055;
      L     "MD654";
      T     DB21.DBD 234;
M055: NOP   0;
      A     L 8.1;
      A(;
      L     DB7.DBB 375;
      L     13;
      ==I;
      );
      =     L 8.2;
      A     L 8.2;
      A     DB21.DBX 394.0;
      =     L 8.3;
      A     L 8.3;
      JNB   M056;
      L     "MD650";
      T     DB21.DBD 238;
M056: NOP   0;
      A     L 8.3;
      JNB   M057;
      L     "MD654";
      T     DB21.DBD 242;
M057: NOP   0;
      A     L 8.2;
      AN    DB21.DBX 394.0;
      =     L 8.3;
      A     L 8.3;
      JNB   M058;
      L     "MD650";
      T     DB21.DBD 246;
M058: NOP   0;
      A     L 8.3;
      JNB   M059;
      L     "MD654";
      T     DB21.DBD 250;
M059: NOP   0;
      A     L 8.1;
      A(;
      L     DB7.DBB 375;
      L     14;
      ==I;
      );
      =     L 8.2;
      A     L 8.2;
      JNB   M060;
      L     "MD650";
      T     DB21.DBD 396;
M060: NOP   0;
      A     L 8.2;
      JNB   M061;
      L     "MD654";
      T     DB21.DBD 400;
M061: NOP   0;
      A     L 8.1;
      JNB   M062;
      L     6;
      T     DB7.DBW 364;
M062: NOP   0;
      A     L 8.1;
      JNB   M063;
      L     "MD650";
      T     "MD588";
M063: NOP   0;
      A     L 8.1;
      JNB   M064;
      L     "MD654";
      T     "MD592";
M064: NOP   0;
      A     L 8.1;
      BLD   102;
      S     "M75.1";
      A     L 8.1;
      FP    "M1004.5";
      JNB   M065;
      L     5;
      T     DB7.DBW 364;
M065: NOP   0;
      A     L 8.0;
      BLD   102;
      R     "M75.0";
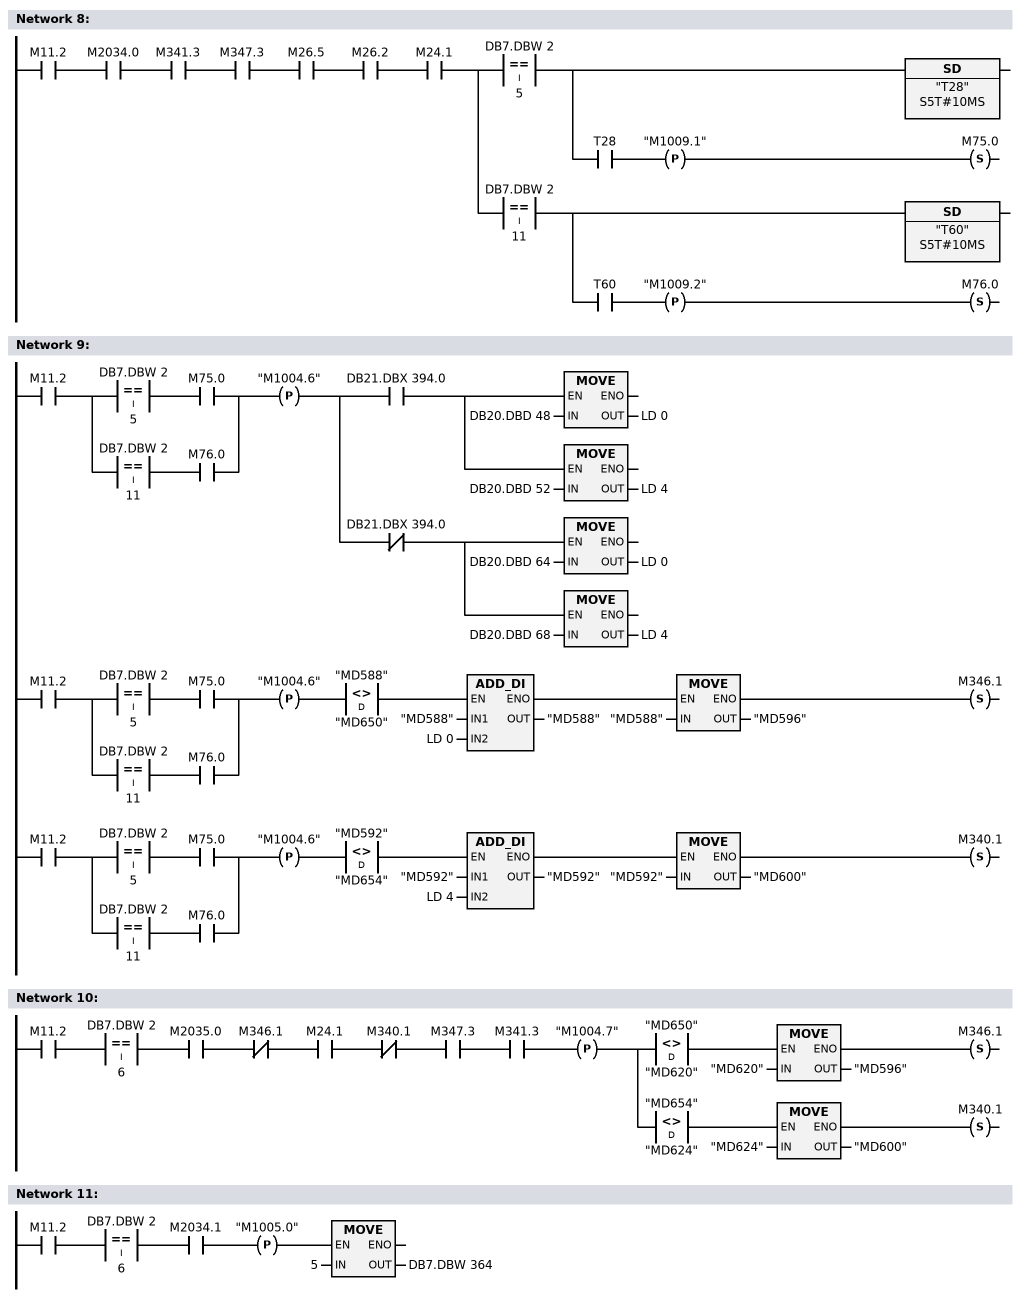
NETWORK
TITLE =
      A     "M11.2";
      A     "M2034.0";
      A     "M341.3";
      A     "M347.3";
      A     "M26.5";
      A     "M26.2";
      A     "M24.1";
      =     L 8.0;
      A     L 8.0;
      A(;
      L     DB7.DBW 2;
      L     5;
      ==I;
      );
      =     L 8.1;
      A     L 8.1;
      BLD   102;
      L     S5T#10MS;
      SD    "T28";
      A     L 8.1;
      A     "T28";
      FP    "M1009.1";
      S     "M75.0";
      A     L 8.0;
      A(;
      L     DB7.DBW 2;
      L     11;
      ==I;
      );
      =     L 8.1;
      A     L 8.1;
      BLD   102;
      L     S5T#10MS;
      SD    "T60";
      A     L 8.1;
      A     "T60";
      FP    "M1009.2";
      S     "M76.0";
NETWORK
TITLE =
      A     "M11.2";
      A(;
      A(;
      L     DB7.DBW 2;
      L     5;
      ==I;
      );
      A     "M75.0";
      O;
      A(;
      L     DB7.DBW 2;
      L     11;
      ==I;
      );
      A     "M76.0";
      );
      FP    "M1004.6";
      =     L 8.0;
      A     L 8.0;
      A     DB21.DBX 394.0;
      =     L 8.1;
      A     L 8.1;
      JNB   M066;
      L     DB20.DBD 48;
      T     LD 0;
M066: NOP   0;
      A     L 8.1;
      JNB   M067;
      L     DB20.DBD 52;
      T     LD 4;
M067: NOP   0;
      A     L 8.0;
      AN    DB21.DBX 394.0;
      =     L 8.1;
      A     L 8.1;
      JNB   M068;
      L     DB20.DBD 64;
      T     LD 0;
M068: NOP   0;
      A     L 8.1;
      JNB   M069;
      L     DB20.DBD 68;
      T     LD 4;
M069: NOP   0;
      A(;
      A     L 8.0;
      A(;
      L     "MD588";
      L     "MD650";
      <>D;
      );
      JNB   M070;
      L     "MD588";
      L     LD 0;
      +D;
      T     "MD588";
      AN    OV;
      SAVE;
      CLR;
M070: A     BR;
      );
      JNB   M071;
      L     "MD588";
      T     "MD596";
      SET;
      SAVE;
      CLR;
M071: A     BR;
      S     "M346.1";
      A(;
      A     L 8.0;
      A(;
      L     "MD592";
      L     "MD654";
      <>D;
      );
      JNB   M072;
      L     "MD592";
      L     LD 4;
      +D;
      T     "MD592";
      AN    OV;
      SAVE;
      CLR;
M072: A     BR;
      );
      JNB   M073;
      L     "MD592";
      T     "MD600";
      SET;
      SAVE;
      CLR;
M073: A     BR;
      S     "M340.1";
NETWORK
TITLE =
      A     "M11.2";
      A(;
      L     DB7.DBW 2;
      L     6;
      ==I;
      );
      A     "M2035.0";
      AN    "M346.1";
      A     "M24.1";
      AN    "M340.1";
      A     "M347.3";
      A     "M341.3";
      FP    "M1004.7";
      =     L 8.0;
      A     L 8.0;
      A(;
      L     "MD650";
      L     "MD620";
      <>D;
      );
      JNB   M074;
      L     "MD620";
      T     "MD596";
      SET;
      SAVE;
      CLR;
M074: A     BR;
      S     "M346.1";
      A     L 8.0;
      A(;
      L     "MD654";
      L     "MD624";
      <>D;
      );
      JNB   M075;
      L     "MD624";
      T     "MD600";
      SET;
      SAVE;
      CLR;
M075: A     BR;
      S     "M340.1";
NETWORK
TITLE =
      A     "M11.2";
      A(;
      L     DB7.DBW 2;
      L     6;
      ==I;
      );
      A     "M2034.1";
      FP    "M1005.0";
      JNB   M076;
      L     5;
      T     DB7.DBW 364;
M076: NOP   0;
END_FUNCTION

FUNCTION "FC51 - TYPE TOOL" : VOID	// FC 51
VERSION : 0.1
BEGIN
// (block stored without names or comments; labels and parameter names are numbered)
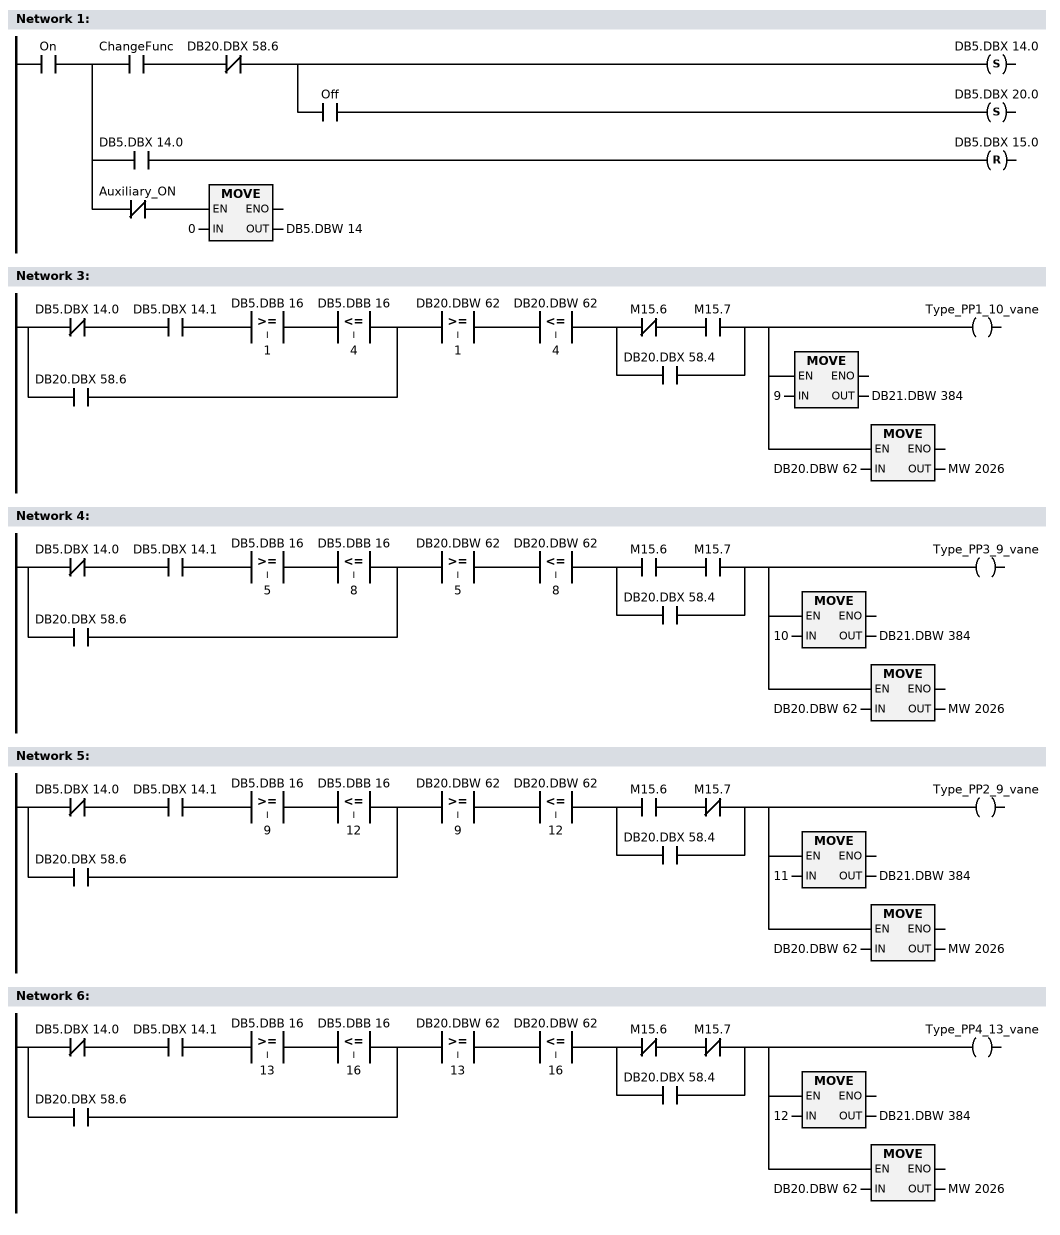
NETWORK
TITLE =
      A     "On";
      =     L 0.0;
      A     L 0.0;
      A     "ChangeFunc";
      AN    DB20.DBX 58.6;
      =     L 0.1;
      A     L 0.1;
      BLD   102;
      S     DB5.DBX 14.0;
      A     L 0.1;
      A     "Off";
      S     DB5.DBX 20.0;
      A     L 0.0;
      A     DB5.DBX 14.0;
      R     DB5.DBX 15.0;
      A     L 0.0;
      AN    "Auxiliary_ON";
      JNB   M001;
      L     0;
      T     DB5.DBW 14;
M001: NOP   0;
NETWORK
TITLE =
NETWORK
TITLE =
      A(;
      AN    DB5.DBX 14.0;
      A     DB5.DBX 14.1;
      A(;
      L     DB5.DBB 16;
      L     1;
      >=I;
      );
      A(;
      L     DB5.DBB 16;
      L     4;
      <=I;
      );
      O     DB20.DBX 58.6;
      );
      A(;
      L     DB20.DBW 62;
      L     1;
      >=I;
      );
      A(;
      L     DB20.DBW 62;
      L     4;
      <=I;
      );
      A(;
      AN    "M15.6";
      A     "M15.7";
      O     DB20.DBX 58.4;
      );
      =     L 0.0;
      A     L 0.0;
      BLD   102;
      =     "Type_PP1_10_vane";
      A     L 0.0;
      JNB   M002;
      L     9;
      T     DB21.DBW 384;
M002: NOP   0;
      A     L 0.0;
      JNB   M003;
      L     DB20.DBW 62;
      T     MW 2026;
M003: NOP   0;
NETWORK
TITLE =
      A(;
      AN    DB5.DBX 14.0;
      A     DB5.DBX 14.1;
      A(;
      L     DB5.DBB 16;
      L     5;
      >=I;
      );
      A(;
      L     DB5.DBB 16;
      L     8;
      <=I;
      );
      O     DB20.DBX 58.6;
      );
      A(;
      L     DB20.DBW 62;
      L     5;
      >=I;
      );
      A(;
      L     DB20.DBW 62;
      L     8;
      <=I;
      );
      A(;
      A     "M15.6";
      A     "M15.7";
      O     DB20.DBX 58.4;
      );
      =     L 0.0;
      A     L 0.0;
      BLD   102;
      =     "Type_PP3_9_vane";
      A     L 0.0;
      JNB   M004;
      L     10;
      T     DB21.DBW 384;
M004: NOP   0;
      A     L 0.0;
      JNB   M005;
      L     DB20.DBW 62;
      T     MW 2026;
M005: NOP   0;
NETWORK
TITLE =
      A(;
      AN    DB5.DBX 14.0;
      A     DB5.DBX 14.1;
      A(;
      L     DB5.DBB 16;
      L     9;
      >=I;
      );
      A(;
      L     DB5.DBB 16;
      L     12;
      <=I;
      );
      O     DB20.DBX 58.6;
      );
      A(;
      L     DB20.DBW 62;
      L     9;
      >=I;
      );
      A(;
      L     DB20.DBW 62;
      L     12;
      <=I;
      );
      A(;
      A     "M15.6";
      AN    "M15.7";
      O     DB20.DBX 58.4;
      );
      =     L 0.0;
      A     L 0.0;
      BLD   102;
      =     "Type_PP2_9_vane";
      A     L 0.0;
      JNB   M006;
      L     11;
      T     DB21.DBW 384;
M006: NOP   0;
      A     L 0.0;
      JNB   M007;
      L     DB20.DBW 62;
      T     MW 2026;
M007: NOP   0;
NETWORK
TITLE =
      A(;
      AN    DB5.DBX 14.0;
      A     DB5.DBX 14.1;
      A(;
      L     DB5.DBB 16;
      L     13;
      >=I;
      );
      A(;
      L     DB5.DBB 16;
      L     16;
      <=I;
      );
      O     DB20.DBX 58.6;
      );
      A(;
      L     DB20.DBW 62;
      L     13;
      >=I;
      );
      A(;
      L     DB20.DBW 62;
      L     16;
      <=I;
      );
      A(;
      AN    "M15.6";
      AN    "M15.7";
      O     DB20.DBX 58.4;
      );
      =     L 0.0;
      A     L 0.0;
      BLD   102;
      =     "Type_PP4_13_vane";
      A     L 0.0;
      JNB   M008;
      L     12;
      T     DB21.DBW 384;
M008: NOP   0;
      A     L 0.0;
      JNB   M009;
      L     DB20.DBW 62;
      T     MW 2026;
M009: NOP   0;
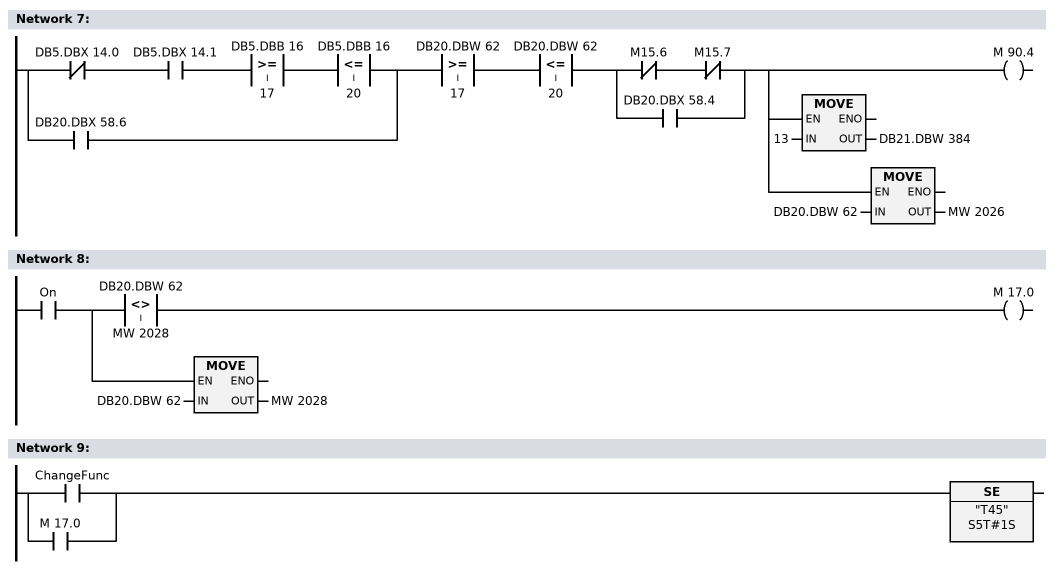
NETWORK
TITLE =
      A(;
      AN    DB5.DBX 14.0;
      A     DB5.DBX 14.1;
      A(;
      L     DB5.DBB 16;
      L     17;
      >=I;
      );
      A(;
      L     DB5.DBB 16;
      L     20;
      <=I;
      );
      O     DB20.DBX 58.6;
      );
      A(;
      L     DB20.DBW 62;
      L     17;
      >=I;
      );
      A(;
      L     DB20.DBW 62;
      L     20;
      <=I;
      );
      A(;
      AN    "M15.6";
      AN    "M15.7";
      O     DB20.DBX 58.4;
      );
      =     L 0.0;
      A     L 0.0;
      BLD   102;
      =     M 90.4;
      A     L 0.0;
      JNB   M010;
      L     13;
      T     DB21.DBW 384;
M010: NOP   0;
      A     L 0.0;
      JNB   M011;
      L     DB20.DBW 62;
      T     MW 2026;
M011: NOP   0;
NETWORK
TITLE =
      A     "On";
      =     L 0.0;
      A     L 0.0;
      A(;
      L     DB20.DBW 62;
      L     MW 2028;
      <>I;
      );
      =     M 17.0;
      A     L 0.0;
      JNB   M012;
      L     DB20.DBW 62;
      T     MW 2028;
M012: NOP   0;
NETWORK
TITLE =
      O     "ChangeFunc";
      O     M 17.0;
      L     S5T#1S;
      SE    "T45";
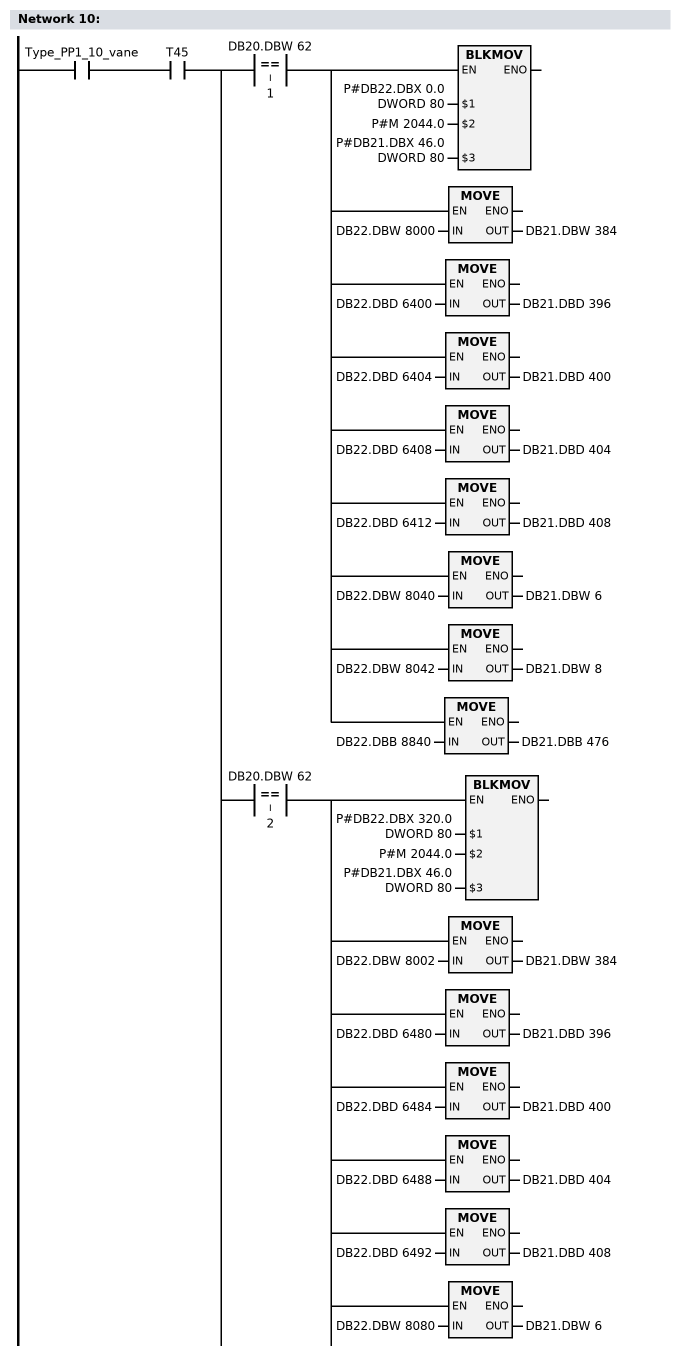
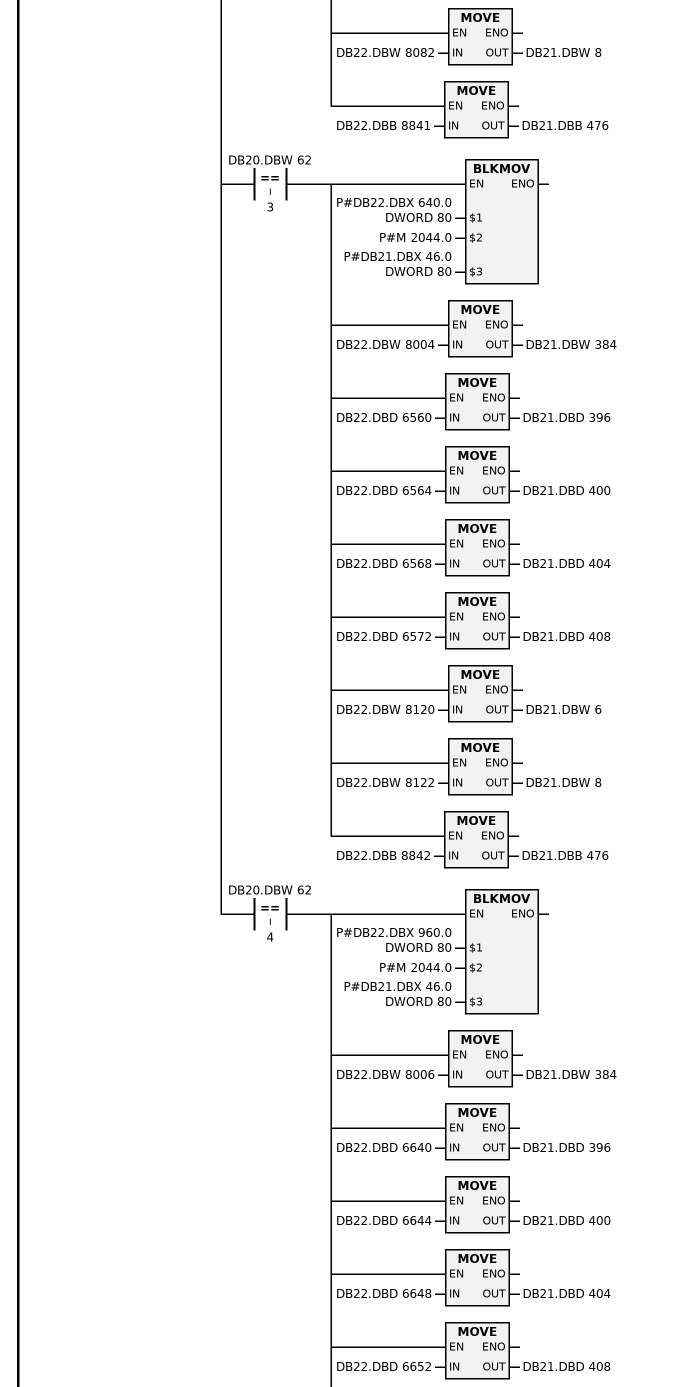
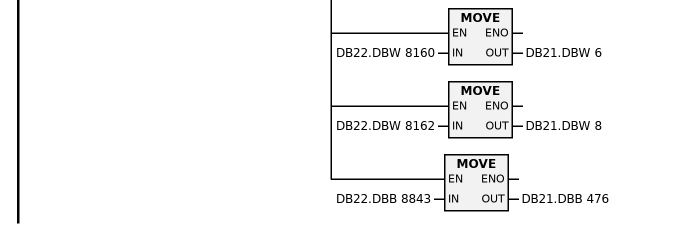
NETWORK
TITLE =
      A     "Type_PP1_10_vane";
      A     "T45";
      =     L 0.0;
      A     L 0.0;
      A(;
      L     DB20.DBW 62;
      L     1;
      ==I;
      );
      =     L 0.1;
      A     L 0.1;
      JNB   M013;
      CALL  "BLKMOV" (
           $1                       := P#DB22.DBX 0.0 DWORD 80,
           $2                       := P#M 2044.0,
           $3                       := P#DB21.DBX 46.0 DWORD 80);
M013: NOP   0;
      A     L 0.1;
      JNB   M014;
      L     DB22.DBW 8000;
      T     DB21.DBW 384;
M014: NOP   0;
      A     L 0.1;
      JNB   M015;
      L     DB22.DBD 6400;
      T     DB21.DBD 396;
M015: NOP   0;
      A     L 0.1;
      JNB   M016;
      L     DB22.DBD 6404;
      T     DB21.DBD 400;
M016: NOP   0;
      A     L 0.1;
      JNB   M017;
      L     DB22.DBD 6408;
      T     DB21.DBD 404;
M017: NOP   0;
      A     L 0.1;
      JNB   M018;
      L     DB22.DBD 6412;
      T     DB21.DBD 408;
M018: NOP   0;
      A     L 0.1;
      JNB   M019;
      L     DB22.DBW 8040;
      T     DB21.DBW 6;
M019: NOP   0;
      A     L 0.1;
      JNB   M020;
      L     DB22.DBW 8042;
      T     DB21.DBW 8;
M020: NOP   0;
      A     L 0.1;
      JNB   M021;
      L     DB22.DBB 8840;
      T     DB21.DBB 476;
M021: NOP   0;
      A     L 0.0;
      A(;
      L     DB20.DBW 62;
      L     2;
      ==I;
      );
      =     L 0.1;
      A     L 0.1;
      JNB   M022;
      CALL  "BLKMOV" (
           $1                       := P#DB22.DBX 320.0 DWORD 80,
           $2                       := P#M 2044.0,
           $3                       := P#DB21.DBX 46.0 DWORD 80);
M022: NOP   0;
      A     L 0.1;
      JNB   M023;
      L     DB22.DBW 8002;
      T     DB21.DBW 384;
M023: NOP   0;
      A     L 0.1;
      JNB   M024;
      L     DB22.DBD 6480;
      T     DB21.DBD 396;
M024: NOP   0;
      A     L 0.1;
      JNB   M025;
      L     DB22.DBD 6484;
      T     DB21.DBD 400;
M025: NOP   0;
      A     L 0.1;
      JNB   M026;
      L     DB22.DBD 6488;
      T     DB21.DBD 404;
M026: NOP   0;
      A     L 0.1;
      JNB   M027;
      L     DB22.DBD 6492;
      T     DB21.DBD 408;
M027: NOP   0;
      A     L 0.1;
      JNB   M028;
      L     DB22.DBW 8080;
      T     DB21.DBW 6;
M028: NOP   0;
      A     L 0.1;
      JNB   M029;
      L     DB22.DBW 8082;
      T     DB21.DBW 8;
M029: NOP   0;
      A     L 0.1;
      JNB   M030;
      L     DB22.DBB 8841;
      T     DB21.DBB 476;
M030: NOP   0;
      A     L 0.0;
      A(;
      L     DB20.DBW 62;
      L     3;
      ==I;
      );
      =     L 0.1;
      A     L 0.1;
      JNB   M031;
      CALL  "BLKMOV" (
           $1                       := P#DB22.DBX 640.0 DWORD 80,
           $2                       := P#M 2044.0,
           $3                       := P#DB21.DBX 46.0 DWORD 80);
M031: NOP   0;
      A     L 0.1;
      JNB   M032;
      L     DB22.DBW 8004;
      T     DB21.DBW 384;
M032: NOP   0;
      A     L 0.1;
      JNB   M033;
      L     DB22.DBD 6560;
      T     DB21.DBD 396;
M033: NOP   0;
      A     L 0.1;
      JNB   M034;
      L     DB22.DBD 6564;
      T     DB21.DBD 400;
M034: NOP   0;
      A     L 0.1;
      JNB   M035;
      L     DB22.DBD 6568;
      T     DB21.DBD 404;
M035: NOP   0;
      A     L 0.1;
      JNB   M036;
      L     DB22.DBD 6572;
      T     DB21.DBD 408;
M036: NOP   0;
      A     L 0.1;
      JNB   M037;
      L     DB22.DBW 8120;
      T     DB21.DBW 6;
M037: NOP   0;
      A     L 0.1;
      JNB   M038;
      L     DB22.DBW 8122;
      T     DB21.DBW 8;
M038: NOP   0;
      A     L 0.1;
      JNB   M039;
      L     DB22.DBB 8842;
      T     DB21.DBB 476;
M039: NOP   0;
      A     L 0.0;
      A(;
      L     DB20.DBW 62;
      L     4;
      ==I;
      );
      =     L 0.1;
      A     L 0.1;
      JNB   M040;
      CALL  "BLKMOV" (
           $1                       := P#DB22.DBX 960.0 DWORD 80,
           $2                       := P#M 2044.0,
           $3                       := P#DB21.DBX 46.0 DWORD 80);
M040: NOP   0;
      A     L 0.1;
      JNB   M041;
      L     DB22.DBW 8006;
      T     DB21.DBW 384;
M041: NOP   0;
      A     L 0.1;
      JNB   M042;
      L     DB22.DBD 6640;
      T     DB21.DBD 396;
M042: NOP   0;
      A     L 0.1;
      JNB   M043;
      L     DB22.DBD 6644;
      T     DB21.DBD 400;
M043: NOP   0;
      A     L 0.1;
      JNB   M044;
      L     DB22.DBD 6648;
      T     DB21.DBD 404;
M044: NOP   0;
      A     L 0.1;
      JNB   M045;
      L     DB22.DBD 6652;
      T     DB21.DBD 408;
M045: NOP   0;
      A     L 0.1;
      JNB   M046;
      L     DB22.DBW 8160;
      T     DB21.DBW 6;
M046: NOP   0;
      A     L 0.1;
      JNB   M047;
      L     DB22.DBW 8162;
      T     DB21.DBW 8;
M047: NOP   0;
      A     L 0.1;
      JNB   M048;
      L     DB22.DBB 8843;
      T     DB21.DBB 476;
M048: NOP   0;
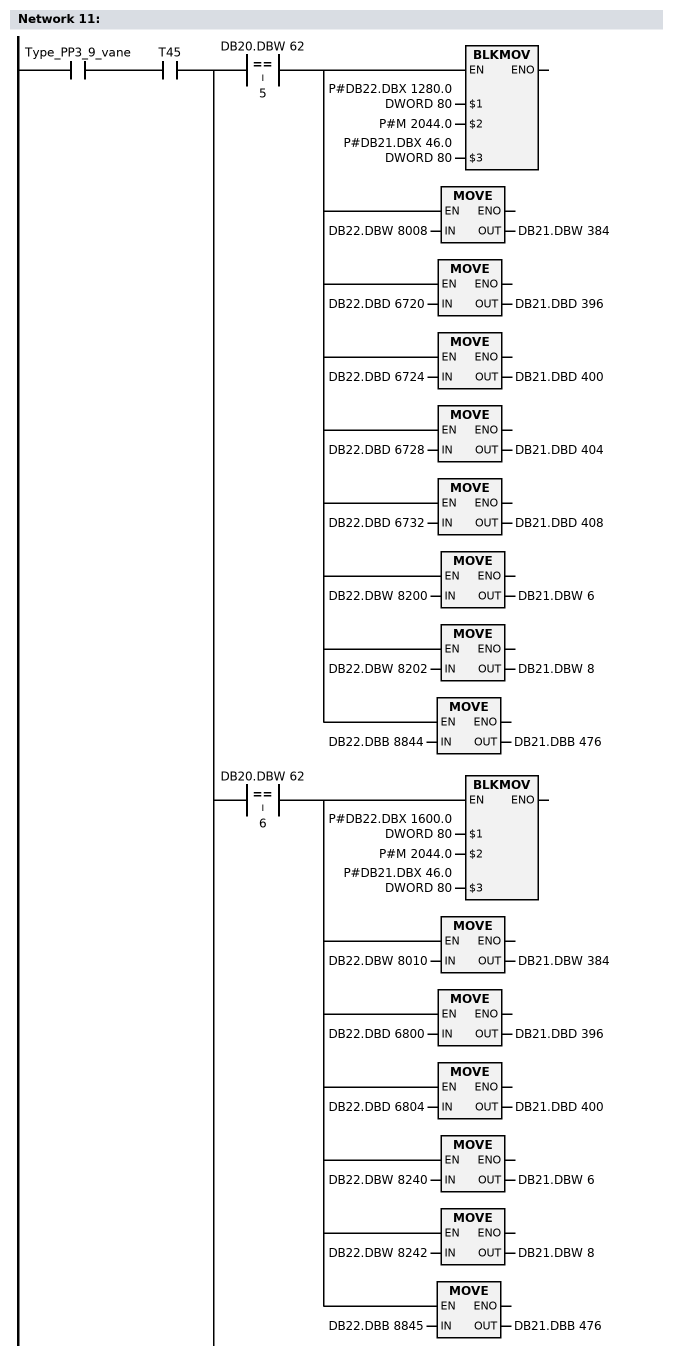
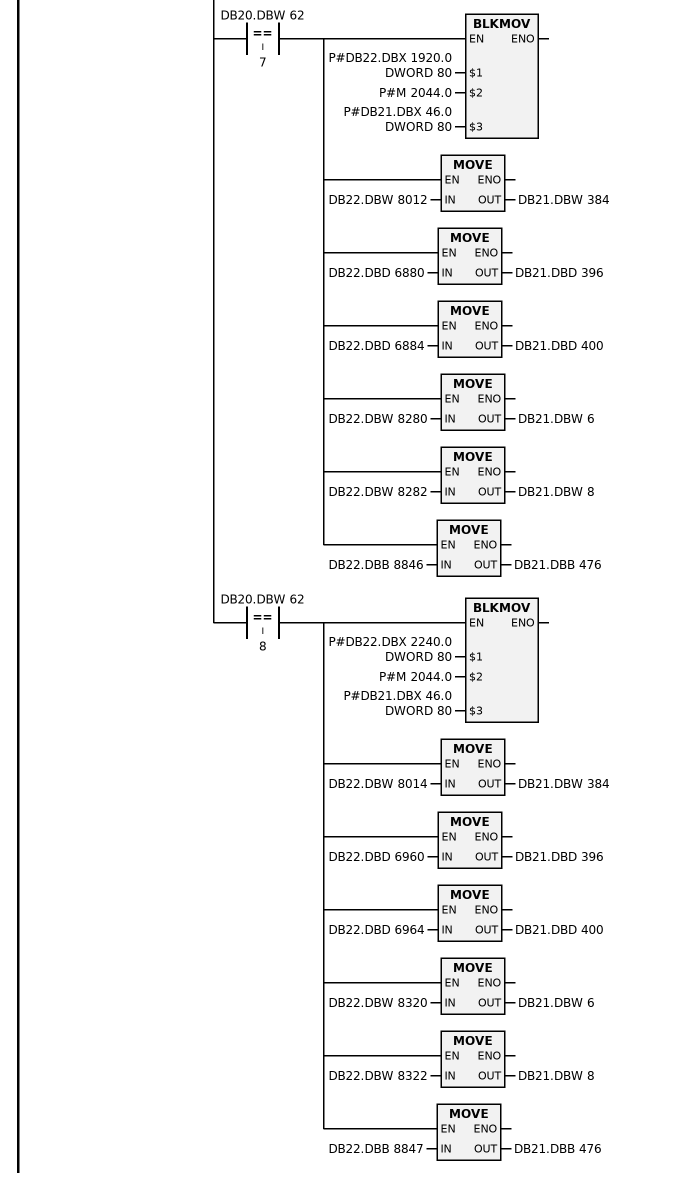
NETWORK
TITLE =
      A     "Type_PP3_9_vane";
      A     "T45";
      =     L 0.0;
      A     L 0.0;
      A(;
      L     DB20.DBW 62;
      L     5;
      ==I;
      );
      =     L 0.1;
      A     L 0.1;
      JNB   M049;
      CALL  "BLKMOV" (
           $1                       := P#DB22.DBX 1280.0 DWORD 80,
           $2                       := P#M 2044.0,
           $3                       := P#DB21.DBX 46.0 DWORD 80);
M049: NOP   0;
      A     L 0.1;
      JNB   M050;
      L     DB22.DBW 8008;
      T     DB21.DBW 384;
M050: NOP   0;
      A     L 0.1;
      JNB   M051;
      L     DB22.DBD 6720;
      T     DB21.DBD 396;
M051: NOP   0;
      A     L 0.1;
      JNB   M052;
      L     DB22.DBD 6724;
      T     DB21.DBD 400;
M052: NOP   0;
      A     L 0.1;
      JNB   M053;
      L     DB22.DBD 6728;
      T     DB21.DBD 404;
M053: NOP   0;
      A     L 0.1;
      JNB   M054;
      L     DB22.DBD 6732;
      T     DB21.DBD 408;
M054: NOP   0;
      A     L 0.1;
      JNB   M055;
      L     DB22.DBW 8200;
      T     DB21.DBW 6;
M055: NOP   0;
      A     L 0.1;
      JNB   M056;
      L     DB22.DBW 8202;
      T     DB21.DBW 8;
M056: NOP   0;
      A     L 0.1;
      JNB   M057;
      L     DB22.DBB 8844;
      T     DB21.DBB 476;
M057: NOP   0;
      A     L 0.0;
      A(;
      L     DB20.DBW 62;
      L     6;
      ==I;
      );
      =     L 0.1;
      A     L 0.1;
      JNB   M058;
      CALL  "BLKMOV" (
           $1                       := P#DB22.DBX 1600.0 DWORD 80,
           $2                       := P#M 2044.0,
           $3                       := P#DB21.DBX 46.0 DWORD 80);
M058: NOP   0;
      A     L 0.1;
      JNB   M059;
      L     DB22.DBW 8010;
      T     DB21.DBW 384;
M059: NOP   0;
      A     L 0.1;
      JNB   M060;
      L     DB22.DBD 6800;
      T     DB21.DBD 396;
M060: NOP   0;
      A     L 0.1;
      JNB   M061;
      L     DB22.DBD 6804;
      T     DB21.DBD 400;
M061: NOP   0;
      A     L 0.1;
      JNB   M062;
      L     DB22.DBW 8240;
      T     DB21.DBW 6;
M062: NOP   0;
      A     L 0.1;
      JNB   M063;
      L     DB22.DBW 8242;
      T     DB21.DBW 8;
M063: NOP   0;
      A     L 0.1;
      JNB   M064;
      L     DB22.DBB 8845;
      T     DB21.DBB 476;
M064: NOP   0;
      A     L 0.0;
      A(;
      L     DB20.DBW 62;
      L     7;
      ==I;
      );
      =     L 0.1;
      A     L 0.1;
      JNB   M065;
      CALL  "BLKMOV" (
           $1                       := P#DB22.DBX 1920.0 DWORD 80,
           $2                       := P#M 2044.0,
           $3                       := P#DB21.DBX 46.0 DWORD 80);
M065: NOP   0;
      A     L 0.1;
      JNB   M066;
      L     DB22.DBW 8012;
      T     DB21.DBW 384;
M066: NOP   0;
      A     L 0.1;
      JNB   M067;
      L     DB22.DBD 6880;
      T     DB21.DBD 396;
M067: NOP   0;
      A     L 0.1;
      JNB   M068;
      L     DB22.DBD 6884;
      T     DB21.DBD 400;
M068: NOP   0;
      A     L 0.1;
      JNB   M069;
      L     DB22.DBW 8280;
      T     DB21.DBW 6;
M069: NOP   0;
      A     L 0.1;
      JNB   M070;
      L     DB22.DBW 8282;
      T     DB21.DBW 8;
M070: NOP   0;
      A     L 0.1;
      JNB   M071;
      L     DB22.DBB 8846;
      T     DB21.DBB 476;
M071: NOP   0;
      A     L 0.0;
      A(;
      L     DB20.DBW 62;
      L     8;
      ==I;
      );
      =     L 0.1;
      A     L 0.1;
      JNB   M072;
      CALL  "BLKMOV" (
           $1                       := P#DB22.DBX 2240.0 DWORD 80,
           $2                       := P#M 2044.0,
           $3                       := P#DB21.DBX 46.0 DWORD 80);
M072: NOP   0;
      A     L 0.1;
      JNB   M073;
      L     DB22.DBW 8014;
      T     DB21.DBW 384;
M073: NOP   0;
      A     L 0.1;
      JNB   M074;
      L     DB22.DBD 6960;
      T     DB21.DBD 396;
M074: NOP   0;
      A     L 0.1;
      JNB   M075;
      L     DB22.DBD 6964;
      T     DB21.DBD 400;
M075: NOP   0;
      A     L 0.1;
      JNB   M076;
      L     DB22.DBW 8320;
      T     DB21.DBW 6;
M076: NOP   0;
      A     L 0.1;
      JNB   M077;
      L     DB22.DBW 8322;
      T     DB21.DBW 8;
M077: NOP   0;
      A     L 0.1;
      JNB   M078;
      L     DB22.DBB 8847;
      T     DB21.DBB 476;
M078: NOP   0;
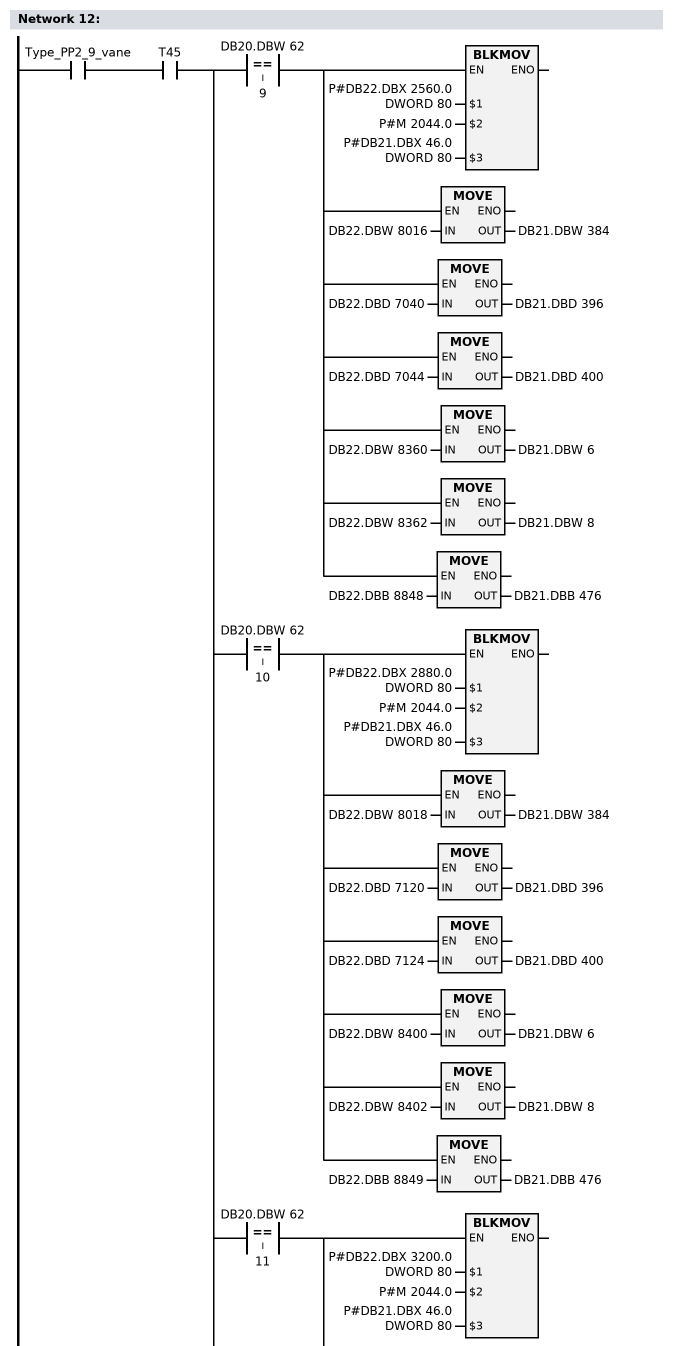
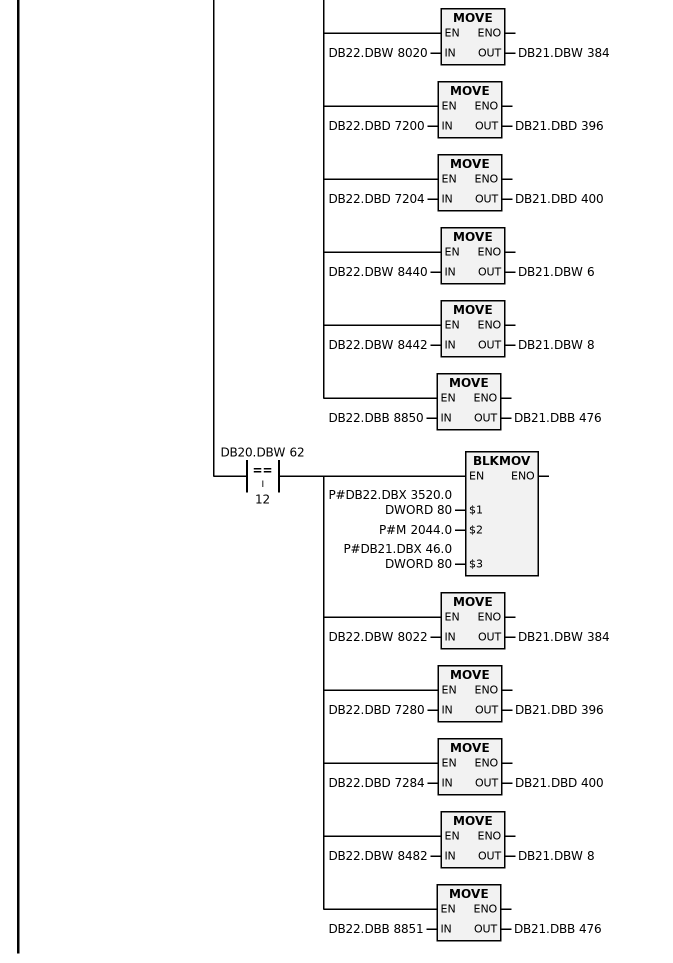
NETWORK
TITLE =
      A     "Type_PP2_9_vane";
      A     "T45";
      =     L 0.0;
      A     L 0.0;
      A(;
      L     DB20.DBW 62;
      L     9;
      ==I;
      );
      =     L 0.1;
      A     L 0.1;
      JNB   M079;
      CALL  "BLKMOV" (
           $1                       := P#DB22.DBX 2560.0 DWORD 80,
           $2                       := P#M 2044.0,
           $3                       := P#DB21.DBX 46.0 DWORD 80);
M079: NOP   0;
      A     L 0.1;
      JNB   M080;
      L     DB22.DBW 8016;
      T     DB21.DBW 384;
M080: NOP   0;
      A     L 0.1;
      JNB   M081;
      L     DB22.DBD 7040;
      T     DB21.DBD 396;
M081: NOP   0;
      A     L 0.1;
      JNB   M082;
      L     DB22.DBD 7044;
      T     DB21.DBD 400;
M082: NOP   0;
      A     L 0.1;
      JNB   M083;
      L     DB22.DBW 8360;
      T     DB21.DBW 6;
M083: NOP   0;
      A     L 0.1;
      JNB   M084;
      L     DB22.DBW 8362;
      T     DB21.DBW 8;
M084: NOP   0;
      A     L 0.1;
      JNB   M085;
      L     DB22.DBB 8848;
      T     DB21.DBB 476;
M085: NOP   0;
      A     L 0.0;
      A(;
      L     DB20.DBW 62;
      L     10;
      ==I;
      );
      =     L 0.1;
      A     L 0.1;
      JNB   M086;
      CALL  "BLKMOV" (
           $1                       := P#DB22.DBX 2880.0 DWORD 80,
           $2                       := P#M 2044.0,
           $3                       := P#DB21.DBX 46.0 DWORD 80);
M086: NOP   0;
      A     L 0.1;
      JNB   M087;
      L     DB22.DBW 8018;
      T     DB21.DBW 384;
M087: NOP   0;
      A     L 0.1;
      JNB   M088;
      L     DB22.DBD 7120;
      T     DB21.DBD 396;
M088: NOP   0;
      A     L 0.1;
      JNB   M089;
      L     DB22.DBD 7124;
      T     DB21.DBD 400;
M089: NOP   0;
      A     L 0.1;
      JNB   M090;
      L     DB22.DBW 8400;
      T     DB21.DBW 6;
M090: NOP   0;
      A     L 0.1;
      JNB   M091;
      L     DB22.DBW 8402;
      T     DB21.DBW 8;
M091: NOP   0;
      A     L 0.1;
      JNB   M092;
      L     DB22.DBB 8849;
      T     DB21.DBB 476;
M092: NOP   0;
      A     L 0.0;
      A(;
      L     DB20.DBW 62;
      L     11;
      ==I;
      );
      =     L 0.1;
      A     L 0.1;
      JNB   M093;
      CALL  "BLKMOV" (
           $1                       := P#DB22.DBX 3200.0 DWORD 80,
           $2                       := P#M 2044.0,
           $3                       := P#DB21.DBX 46.0 DWORD 80);
M093: NOP   0;
      A     L 0.1;
      JNB   M094;
      L     DB22.DBW 8020;
      T     DB21.DBW 384;
M094: NOP   0;
      A     L 0.1;
      JNB   M095;
      L     DB22.DBD 7200;
      T     DB21.DBD 396;
M095: NOP   0;
      A     L 0.1;
      JNB   M096;
      L     DB22.DBD 7204;
      T     DB21.DBD 400;
M096: NOP   0;
      A     L 0.1;
      JNB   M097;
      L     DB22.DBW 8440;
      T     DB21.DBW 6;
M097: NOP   0;
      A     L 0.1;
      JNB   M098;
      L     DB22.DBW 8442;
      T     DB21.DBW 8;
M098: NOP   0;
      A     L 0.1;
      JNB   M099;
      L     DB22.DBB 8850;
      T     DB21.DBB 476;
M099: NOP   0;
      A     L 0.0;
      A(;
      L     DB20.DBW 62;
      L     12;
      ==I;
      );
      =     L 0.1;
      A     L 0.1;
      JNB   M100;
      CALL  "BLKMOV" (
           $1                       := P#DB22.DBX 3520.0 DWORD 80,
           $2                       := P#M 2044.0,
           $3                       := P#DB21.DBX 46.0 DWORD 80);
M100: NOP   0;
      A     L 0.1;
      JNB   M101;
      L     DB22.DBW 8022;
      T     DB21.DBW 384;
M101: NOP   0;
      A     L 0.1;
      JNB   M102;
      L     DB22.DBD 7280;
      T     DB21.DBD 396;
M102: NOP   0;
      A     L 0.1;
      JNB   M103;
      L     DB22.DBD 7284;
      T     DB21.DBD 400;
M103: NOP   0;
      A     L 0.1;
      JNB   M104;
      L     DB22.DBW 8482;
      T     DB21.DBW 8;
M104: NOP   0;
      A     L 0.1;
      JNB   M105;
      L     DB22.DBB 8851;
      T     DB21.DBB 476;
M105: NOP   0;
